// TIA Portal V20 export
FUNCTION_BLOCK "Sequence_1_SepaClamp"   // FB197, LAD
AUTHOR : ERsystem_FA2_DH. Kim
// stored: IsIECCheckEnabled true, MemoryReserve 100, Namespace Unit1.Em7, SetENOAutomatically false
   VAR
      statSelectedJobNumber { ExternalWritable := 'False'} : DInt;   // Evaluated Job Number
      instSequenceLADStatus { ExternalWritable := 'False'} : "LAF_StatusLadSequence";
      instSequenceLADControl { ExternalWritable := 'False'} : "LAF_ControlLadSequence";
      statTonTime { ExternalAccessible := 'False'; ExternalVisible := 'False'; ExternalWritable := 'False'} : Array[0..999] of TON_TIME;
   END_VAR
   VAR_TEMP
      tempCustomerAction : Bool;   // Placeholder for possible actions
      tempDo_nothing_and_wait_for_init : Bool;   // Placeholder for doing nothing
      tempSafeStateCondition : Bool;   // Temp Condition for the equipment module to be in a safe state
      tempIndex : Int;
   END_VAR
   VAR CONSTANT
      STEP_IDLE : DInt := 1;
      STEP_IMMEDIATE_STOP : DInt := 9001;   // Step executed when an immediate stop command is triggered for the sequence (i.e. when unit is in state aborting)
      JOB_1_STEP_01 : DInt := 101;
      JOB_1_STEP_10 : DInt := 110;
      JOB_1_STEP_20 : DInt := 120;
      JOB_1_STEP_30 : DInt := 130;
      JOB_1_STEP_80 : DInt := 180;
      JOB_1_STEP_90 : DInt := 190;
      JOB_2_STEP_01 : DInt := 201;
      JOB_2_STEP_10 : DInt := 210;
      JOB_2_STEP_11 : DInt := 211;
      JOB_2_STEP_20 : DInt := 220;
      JOB_2_STEP_21 : DInt := 221;
      JOB_2_STEP_30 : DInt := 230;
      JOB_2_STEP_40 : DInt := 240;
      JOB_2_STEP_41 : DInt := 241;
      JOB_2_STEP_50 : DInt := 250;
      JOB_2_STEP_51 : DInt := 251;
      JOB_2_STEP_60 : DInt := 260;
      JOB_2_STEP_80 : DInt := 280;
      JOB_2_STEP_90 : DInt := 290;
      JOB_3_STEP_01 : DInt := 301;
      JOB_3_STEP_10 : DInt := 310;
      JOB_3_STEP_11 : DInt := 311;
      JOB_3_STEP_20 : DInt := 320;
      JOB_3_STEP_21 : DInt := 321;
      JOB_3_STEP_22 : DInt := 322;
      JOB_3_STEP_23 : DInt := 323;
      JOB_3_STEP_24 : DInt := 324;
      JOB_3_STEP_30 : DInt := 330;
      JOB_3_STEP_31 : DInt := 331;
      JOB_3_STEP_40 : DInt := 340;
      JOB_3_STEP_80 : DInt := 380;
      JOB_3_STEP_90 : DInt := 390;
      JOB_4_STEP_01 : DInt := 401;
      JOB_4_STEP_10 : DInt := 410;
      JOB_4_STEP_11 : DInt := 411;
      JOB_4_STEP_90 : DInt := 490;
      JOB_5_STEP_01 : DInt := 501;
      JOB_5_STEP_10 : DInt := 510;
      JOB_5_STEP_11 : DInt := 511;
      JOB_5_STEP_20 : DInt := 520;
      JOB_5_STEP_21 : DInt := 521;
      JOB_5_STEP_30 : DInt := 530;
      JOB_5_STEP_90 : DInt := 590;
      JOB_6_STEP_01 : DInt := 601;
      JOB_6_STEP_10 : DInt := 610;
      JOB_6_STEP_11 : DInt := 611;
      JOB_6_STEP_20 : DInt := 620;
      JOB_6_STEP_30 : DInt := 630;
      JOB_6_STEP_90 : DInt := 690;
      JOB_10_STEP_01 : DInt := 1001;
      JOB_10_STEP_10 : DInt := 1010;
      JOB_10_STEP_11 : DInt := 1011;
      JOB_10_STEP_20 : DInt := 1020;
      JOB_10_STEP_90 : DInt := 1090;
      JOB_11_STEP_01 : DInt := 1101;
      JOB_11_STEP_10 : DInt := 1110;
      JOB_11_STEP_20 : DInt := 1120;
      JOB_11_STEP_30 : DInt := 1130;
      JOB_11_STEP_90 : DInt := 1190;
      JOB_12_STEP_01 : DInt := 1201;
      JOB_12_STEP_10 : DInt := 1210;
      JOB_12_STEP_20 : DInt := 1220;
      JOB_12_STEP_30 : DInt := 1230;
      JOB_12_STEP_40 : DInt := 1240;
      JOB_12_STEP_90 : DInt := 1290;
      FALSE : Bool := FALSE;
      TRUE : Bool := TRUE;
   END_VAR
   VAR_TEMP   // added for the SCL form of the ladder/FBD networks
      _w1 : Bool;
      _w2 : Bool;
   END_VAR
BEGIN

REGION Network 1: BLOCK INFO HEADER
   // (company) / (C) Copyright (year)
   // ---------------------------------------------------------------------------------
   // Title:                             (Title of this block)
   // Comment/Function: (that is implemented in the block)
   // Library/Family:           (that the source is dedicated to)
   // Author:                        (department / person in charge / contact)
   // Target System:          (test system with FW version)
   // Engineering:              TIA Portal (SW version)
   // Restrictions:               (OB types, etc.)
   // Requirements:           (hardware, technological package, etc.)
   // ---------------------------------------------------------------------------------
   // Change log table:
   // Version          | Date             | Signature      | Expert in charge  | Changes applied ------------------------|----------------------|-------------------------|--------------------------------|-----------------------
   // 001.000.000 | yyyy-mm-dd | 0x00000000 | (name of expert) | First released version
END_REGION

REGION Network 2: DESCRIPTION
   // This is a template block provided by the Automation Framework. It can be used to create an own project.
   // The Block Info Header is prepared to put in your own data.
   // Description of the block could be added here and the docu created by Code2Docu.
END_REGION

REGION Network 3: ********************* CONTROL *************************
END_REGION

REGION Network 4: Sequence Control
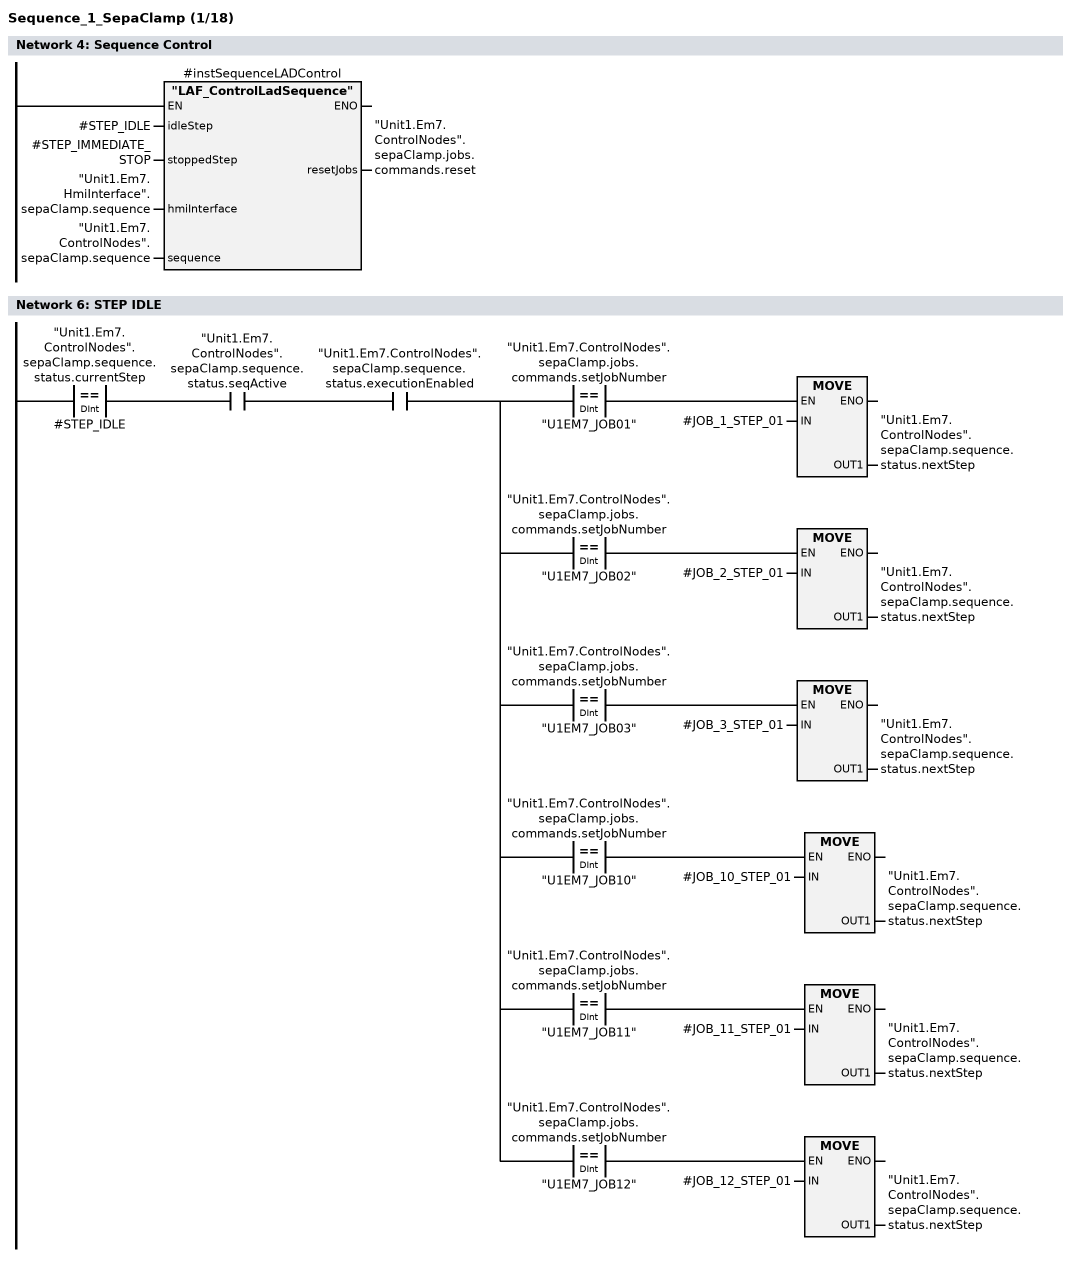
   RUNG wire#powerrail
      #instSequenceLADControl(idleStep := #STEP_IDLE, stoppedStep := #STEP_IMMEDIATE_STOP, hmiInterface := "Unit1.Em7.HmiInterface".sepaClamp.sequence, sequence := "Unit1.Em7.ControlNodes".sepaClamp.sequence, resetJobs => "Unit1.Em7.ControlNodes".sepaClamp.jobs.commands.reset)
   END_RUNG
   // the same network as SCL:
   #instSequenceLADControl(idleStep := #STEP_IDLE,   // "LAF_ControlLadSequence"
                           stoppedStep := #STEP_IMMEDIATE_STOP,
                           hmiInterface := "Unit1.Em7.HmiInterface".sepaClamp.sequence,
                           sequence := "Unit1.Em7.ControlNodes".sepaClamp.sequence,
                           resetJobs => "Unit1.Em7.ControlNodes".sepaClamp.jobs.commands.reset);
END_REGION

REGION Network 5: *************** JOB SELECT **************************
END_REGION

REGION Network 6: STEP IDLE
   RUNG wire#powerrail
      { S7_Templates := "SrcType := DInt" } EQ_Contact(in1 := "Unit1.Em7.ControlNodes".sepaClamp.sequence.status.currentStep, in2 := #STEP_IDLE)
      Contact( "Unit1.Em7.ControlNodes".sepaClamp.sequence.status.seqActive )
      Contact( "Unit1.Em7.ControlNodes".sepaClamp.sequence.status.executionEnabled )
      wire#w1
      { S7_Templates := "SrcType := DInt" } EQ_Contact(in1 := "Unit1.Em7.ControlNodes".sepaClamp.jobs.commands.setJobNumber, in2 := "U1EM7_JOB01")
      Move(in := #JOB_1_STEP_01, out1 => "Unit1.Em7.ControlNodes".sepaClamp.sequence.status.nextStep)
   END_RUNG
   RUNG wire#w1
      { S7_Templates := "SrcType := DInt" } EQ_Contact(in1 := "Unit1.Em7.ControlNodes".sepaClamp.jobs.commands.setJobNumber, in2 := "U1EM7_JOB02")
      Move(in := #JOB_2_STEP_01, out1 => "Unit1.Em7.ControlNodes".sepaClamp.sequence.status.nextStep)
   END_RUNG
   RUNG wire#w1
      { S7_Templates := "SrcType := DInt" } EQ_Contact(in1 := "Unit1.Em7.ControlNodes".sepaClamp.jobs.commands.setJobNumber, in2 := "U1EM7_JOB03")
      Move(in := #JOB_3_STEP_01, out1 => "Unit1.Em7.ControlNodes".sepaClamp.sequence.status.nextStep)
   END_RUNG
   RUNG wire#w1
      { S7_Templates := "SrcType := DInt" } EQ_Contact(in1 := "Unit1.Em7.ControlNodes".sepaClamp.jobs.commands.setJobNumber, in2 := "U1EM7_JOB10")
      Move(in := #JOB_10_STEP_01, out1 => "Unit1.Em7.ControlNodes".sepaClamp.sequence.status.nextStep)
   END_RUNG
   RUNG wire#w1
      { S7_Templates := "SrcType := DInt" } EQ_Contact(in1 := "Unit1.Em7.ControlNodes".sepaClamp.jobs.commands.setJobNumber, in2 := "U1EM7_JOB11")
      Move(in := #JOB_11_STEP_01, out1 => "Unit1.Em7.ControlNodes".sepaClamp.sequence.status.nextStep)
   END_RUNG
   RUNG wire#w1
      { S7_Templates := "SrcType := DInt" } EQ_Contact(in1 := "Unit1.Em7.ControlNodes".sepaClamp.jobs.commands.setJobNumber, in2 := "U1EM7_JOB12")
      Move(in := #JOB_12_STEP_01, out1 => "Unit1.Em7.ControlNodes".sepaClamp.sequence.status.nextStep)
   END_RUNG
   // the same network as SCL:
   #_w1 := ("Unit1.Em7.ControlNodes".sepaClamp.sequence.status.currentStep = #STEP_IDLE) AND "Unit1.Em7.ControlNodes".sepaClamp.sequence.status.seqActive AND "Unit1.Em7.ControlNodes".sepaClamp.sequence.status.executionEnabled;
   IF #_w1 AND ("Unit1.Em7.ControlNodes".sepaClamp.jobs.commands.setJobNumber = "U1EM7_JOB01") THEN
       "Unit1.Em7.ControlNodes".sepaClamp.sequence.status.nextStep := #JOB_1_STEP_01;
   END_IF;
   IF #_w1 AND ("Unit1.Em7.ControlNodes".sepaClamp.jobs.commands.setJobNumber = "U1EM7_JOB02") THEN
       "Unit1.Em7.ControlNodes".sepaClamp.sequence.status.nextStep := #JOB_2_STEP_01;
   END_IF;
   IF #_w1 AND ("Unit1.Em7.ControlNodes".sepaClamp.jobs.commands.setJobNumber = "U1EM7_JOB03") THEN
       "Unit1.Em7.ControlNodes".sepaClamp.sequence.status.nextStep := #JOB_3_STEP_01;
   END_IF;
   IF #_w1 AND ("Unit1.Em7.ControlNodes".sepaClamp.jobs.commands.setJobNumber = "U1EM7_JOB10") THEN
       "Unit1.Em7.ControlNodes".sepaClamp.sequence.status.nextStep := #JOB_10_STEP_01;
   END_IF;
   IF #_w1 AND ("Unit1.Em7.ControlNodes".sepaClamp.jobs.commands.setJobNumber = "U1EM7_JOB11") THEN
       "Unit1.Em7.ControlNodes".sepaClamp.sequence.status.nextStep := #JOB_11_STEP_01;
   END_IF;
   IF #_w1 AND ("Unit1.Em7.ControlNodes".sepaClamp.jobs.commands.setJobNumber = "U1EM7_JOB12") THEN
       "Unit1.Em7.ControlNodes".sepaClamp.sequence.status.nextStep := #JOB_12_STEP_01;
   END_IF;
END_REGION

REGION Network 7: *************** JOB[1] EM HOMING ************************
END_REGION

REGION Network 8: Step[101] : JOB[1] Condition
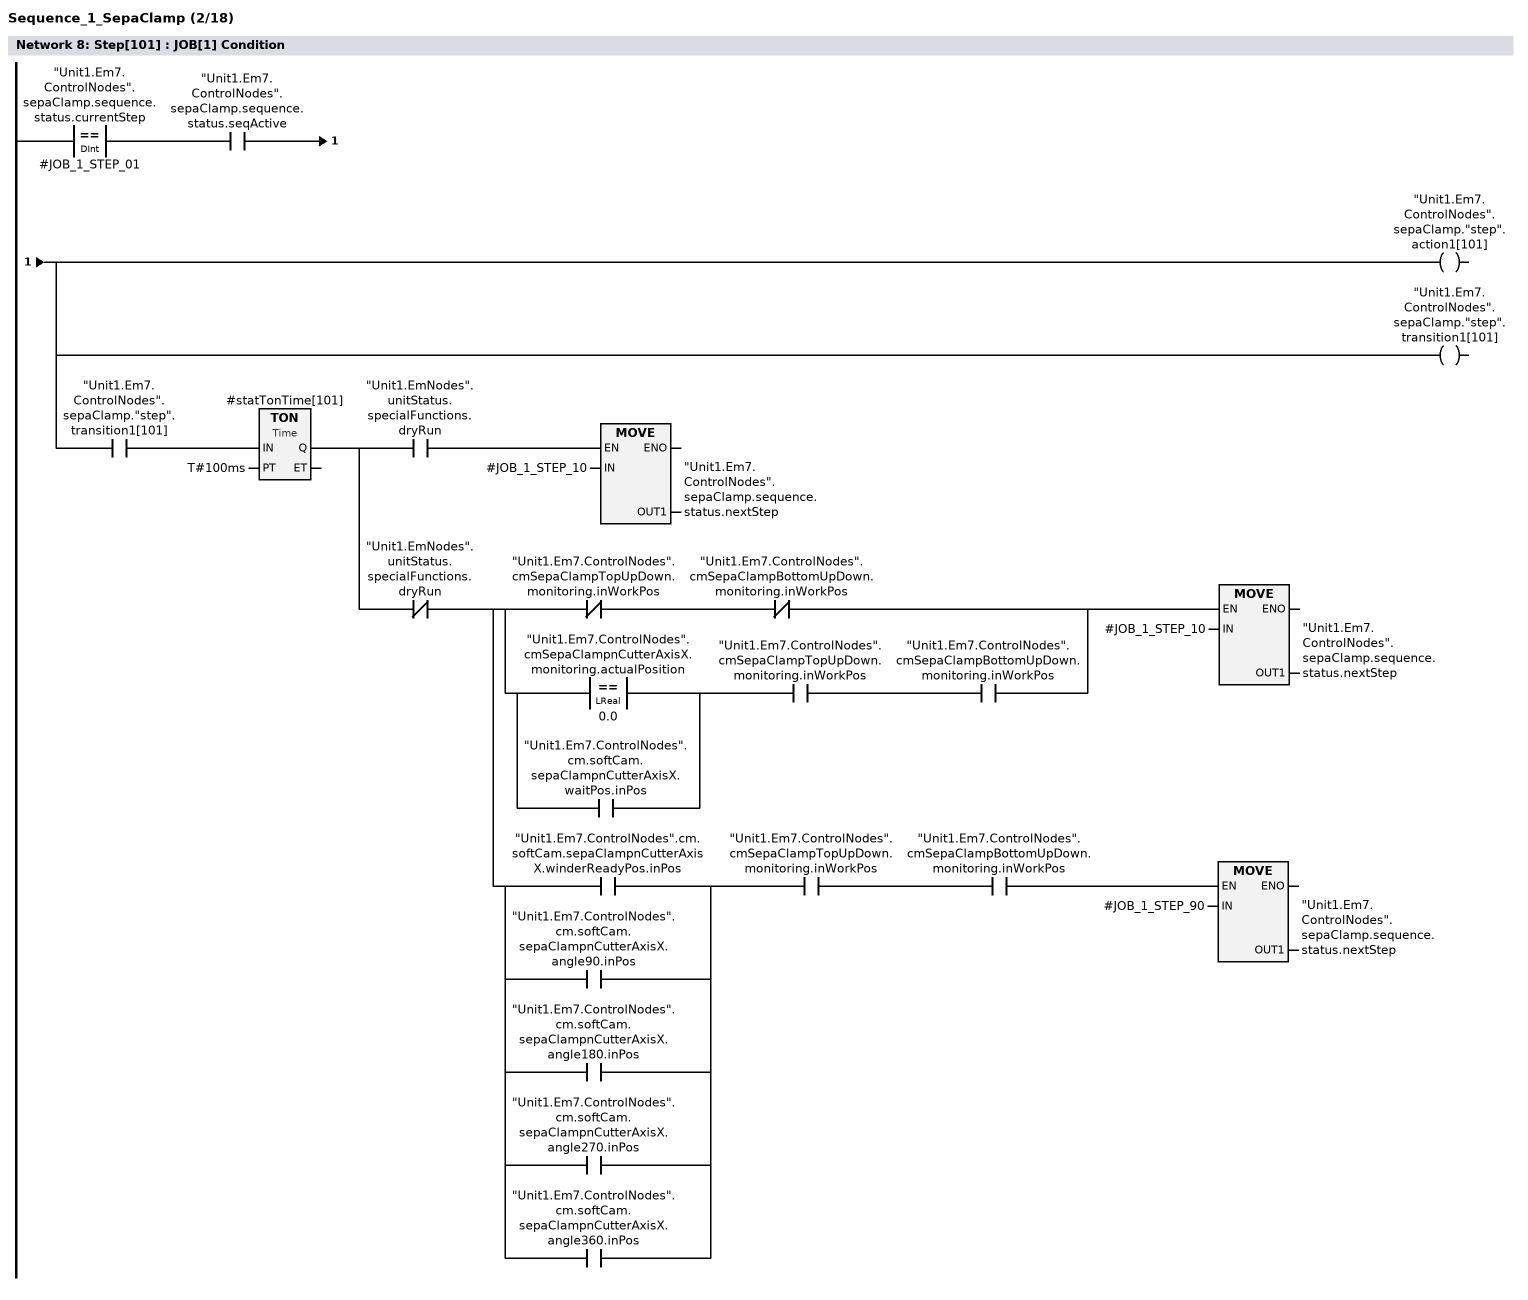
   RUNG wire#powerrail
      { S7_Templates := "SrcType := DInt" } EQ_Contact(in1 := "Unit1.Em7.ControlNodes".sepaClamp.sequence.status.currentStep, in2 := #JOB_1_STEP_01)
      Contact( "Unit1.Em7.ControlNodes".sepaClamp.sequence.status.seqActive )
      wire#w1
      Coil( "Unit1.Em7.ControlNodes".sepaClamp."step".action1[101] )
   END_RUNG
   RUNG wire#w1
      Coil( "Unit1.Em7.ControlNodes".sepaClamp."step".transition1[101] )
   END_RUNG
   RUNG wire#w1
      Contact( "Unit1.Em7.ControlNodes".sepaClamp."step".transition1[101] )
      { S7_Templates := "time_type := Time" } #statTonTime[101].TON(pt := T#100ms, et =>)
      wire#w2
      Contact( "Unit1.EmNodes".unitStatus.specialFunctions.dryRun )
      Move(in := #JOB_1_STEP_10, out1 => "Unit1.Em7.ControlNodes".sepaClamp.sequence.status.nextStep)
   END_RUNG
   RUNG wire#w2
      I_Contact( "Unit1.EmNodes".unitStatus.specialFunctions.dryRun )
      wire#w3
      I_Contact( "Unit1.Em7.ControlNodes".cmSepaClampTopUpDown.monitoring.inWorkPos )
      I_Contact( "Unit1.Em7.ControlNodes".cmSepaClampBottomUpDown.monitoring.inWorkPos )
      wire#w4
      Move(in := #JOB_1_STEP_10, out1 => "Unit1.Em7.ControlNodes".sepaClamp.sequence.status.nextStep)
   END_RUNG
   RUNG wire#w3
      { S7_Templates := "SrcType := LReal" } EQ_Contact(in1 := "Unit1.Em7.ControlNodes".cmSepaClampnCutterAxisX.monitoring.actualPosition, in2 := 0.0)
      wire#w5
      Contact( "Unit1.Em7.ControlNodes".cmSepaClampTopUpDown.monitoring.inWorkPos )
      Contact( "Unit1.Em7.ControlNodes".cmSepaClampBottomUpDown.monitoring.inWorkPos )
   END_RUNG wire#w4
   RUNG wire#w3
      Contact( "Unit1.Em7.ControlNodes".cm.softCam.sepaClampnCutterAxisX.waitPos.inPos )
   END_RUNG wire#w5
   RUNG wire#w3
      Contact( "Unit1.Em7.ControlNodes".cm.softCam.sepaClampnCutterAxisX.winderReadyPos.inPos )
      wire#w6
      Contact( "Unit1.Em7.ControlNodes".cmSepaClampTopUpDown.monitoring.inWorkPos )
      Contact( "Unit1.Em7.ControlNodes".cmSepaClampBottomUpDown.monitoring.inWorkPos )
      Move(in := #JOB_1_STEP_90, out1 => "Unit1.Em7.ControlNodes".sepaClamp.sequence.status.nextStep)
   END_RUNG
   RUNG wire#w3
      Contact( "Unit1.Em7.ControlNodes".cm.softCam.sepaClampnCutterAxisX.angle90.inPos )
   END_RUNG wire#w6
   RUNG wire#w3
      Contact( "Unit1.Em7.ControlNodes".cm.softCam.sepaClampnCutterAxisX.angle180.inPos )
   END_RUNG wire#w6
   RUNG wire#w3
      Contact( "Unit1.Em7.ControlNodes".cm.softCam.sepaClampnCutterAxisX.angle270.inPos )
   END_RUNG wire#w6
   RUNG wire#w3
      Contact( "Unit1.Em7.ControlNodes".cm.softCam.sepaClampnCutterAxisX.angle360.inPos )
   END_RUNG wire#w6
   // the same network as SCL:
   "Unit1.Em7.ControlNodes".sepaClamp."step".action1[101] := ("Unit1.Em7.ControlNodes".sepaClamp.sequence.status.currentStep = #JOB_1_STEP_01) AND "Unit1.Em7.ControlNodes".sepaClamp.sequence.status.seqActive;
   "Unit1.Em7.ControlNodes".sepaClamp."step".transition1[101] := ("Unit1.Em7.ControlNodes".sepaClamp.sequence.status.currentStep = #JOB_1_STEP_01) AND "Unit1.Em7.ControlNodes".sepaClamp.sequence.status.seqActive;
   #statTonTime[101].TON(IN := ("Unit1.Em7.ControlNodes".sepaClamp.sequence.status.currentStep = #JOB_1_STEP_01) AND "Unit1.Em7.ControlNodes".sepaClamp.sequence.status.seqActive AND "Unit1.Em7.ControlNodes".sepaClamp."step".transition1[101],
                         PT := T#100ms);
   IF #statTonTime[101].Q AND "Unit1.EmNodes".unitStatus.specialFunctions.dryRun THEN
       "Unit1.Em7.ControlNodes".sepaClamp.sequence.status.nextStep := #JOB_1_STEP_10;
   END_IF;
   #_w1 := #statTonTime[101].Q AND NOT "Unit1.EmNodes".unitStatus.specialFunctions.dryRun;
   IF #_w1 AND ((NOT "Unit1.Em7.ControlNodes".cmSepaClampTopUpDown.monitoring.inWorkPos AND NOT "Unit1.Em7.ControlNodes".cmSepaClampBottomUpDown.monitoring.inWorkPos) OR ((("Unit1.Em7.ControlNodes".cmSepaClampnCutterAxisX.monitoring.actualPosition = 0.0) OR "Unit1.Em7.ControlNodes".cm.softCam.sepaClampnCutterAxisX.waitPos.inPos) AND "Unit1.Em7.ControlNodes".cmSepaClampTopUpDown.monitoring.inWorkPos AND "Unit1.Em7.ControlNodes".cmSepaClampBottomUpDown.monitoring.inWorkPos)) THEN
       "Unit1.Em7.ControlNodes".sepaClamp.sequence.status.nextStep := #JOB_1_STEP_10;
   END_IF;
   IF #_w1 AND ("Unit1.Em7.ControlNodes".cm.softCam.sepaClampnCutterAxisX.winderReadyPos.inPos OR "Unit1.Em7.ControlNodes".cm.softCam.sepaClampnCutterAxisX.angle90.inPos OR "Unit1.Em7.ControlNodes".cm.softCam.sepaClampnCutterAxisX.angle180.inPos OR "Unit1.Em7.ControlNodes".cm.softCam.sepaClampnCutterAxisX.angle270.inPos OR "Unit1.Em7.ControlNodes".cm.softCam.sepaClampnCutterAxisX.angle360.inPos) AND "Unit1.Em7.ControlNodes".cmSepaClampTopUpDown.monitoring.inWorkPos AND "Unit1.Em7.ControlNodes".cmSepaClampBottomUpDown.monitoring.inWorkPos THEN
       "Unit1.Em7.ControlNodes".sepaClamp.sequence.status.nextStep := #JOB_1_STEP_90;
   END_IF;
END_REGION

REGION Network 9: Step[110] : Cutter Up
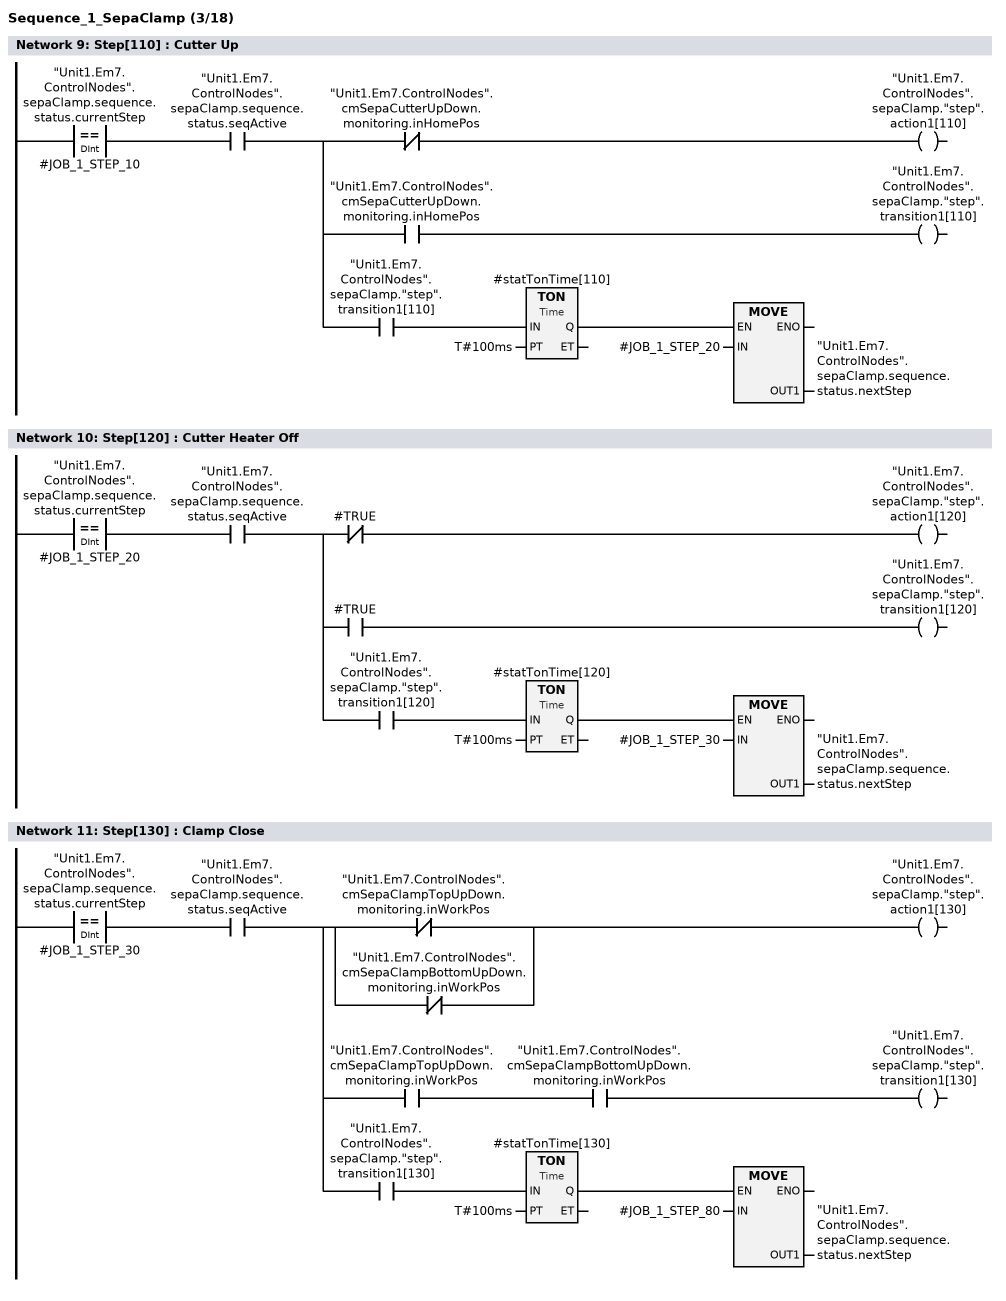
   RUNG wire#powerrail
      { S7_Templates := "SrcType := DInt" } EQ_Contact(in1 := "Unit1.Em7.ControlNodes".sepaClamp.sequence.status.currentStep, in2 := #JOB_1_STEP_10)
      Contact( "Unit1.Em7.ControlNodes".sepaClamp.sequence.status.seqActive )
      wire#w1
      I_Contact( "Unit1.Em7.ControlNodes".cmSepaCutterUpDown.monitoring.inHomePos )
      Coil( "Unit1.Em7.ControlNodes".sepaClamp."step".action1[110] )
   END_RUNG
   RUNG wire#w1
      Contact( "Unit1.Em7.ControlNodes".cmSepaCutterUpDown.monitoring.inHomePos )
      Coil( "Unit1.Em7.ControlNodes".sepaClamp."step".transition1[110] )
   END_RUNG
   RUNG wire#w1
      Contact( "Unit1.Em7.ControlNodes".sepaClamp."step".transition1[110] )
      { S7_Templates := "time_type := Time" } #statTonTime[110].TON(pt := T#100ms, et =>)
      Move(in := #JOB_1_STEP_20, out1 => "Unit1.Em7.ControlNodes".sepaClamp.sequence.status.nextStep)
   END_RUNG
   // the same network as SCL:
   #_w1 := ("Unit1.Em7.ControlNodes".sepaClamp.sequence.status.currentStep = #JOB_1_STEP_10) AND "Unit1.Em7.ControlNodes".sepaClamp.sequence.status.seqActive;
   "Unit1.Em7.ControlNodes".sepaClamp."step".action1[110] := #_w1 AND NOT "Unit1.Em7.ControlNodes".cmSepaCutterUpDown.monitoring.inHomePos;
   "Unit1.Em7.ControlNodes".sepaClamp."step".transition1[110] := #_w1 AND "Unit1.Em7.ControlNodes".cmSepaCutterUpDown.monitoring.inHomePos;
   #statTonTime[110].TON(IN := #_w1 AND "Unit1.Em7.ControlNodes".sepaClamp."step".transition1[110],
                         PT := T#100ms);
   IF #statTonTime[110].Q THEN
       "Unit1.Em7.ControlNodes".sepaClamp.sequence.status.nextStep := #JOB_1_STEP_20;
   END_IF;
END_REGION

REGION Network 10: Step[120] : Cutter Heater Off
   RUNG wire#powerrail
      { S7_Templates := "SrcType := DInt" } EQ_Contact(in1 := "Unit1.Em7.ControlNodes".sepaClamp.sequence.status.currentStep, in2 := #JOB_1_STEP_20)
      Contact( "Unit1.Em7.ControlNodes".sepaClamp.sequence.status.seqActive )
      wire#w1
      I_Contact( #TRUE )
      Coil( "Unit1.Em7.ControlNodes".sepaClamp."step".action1[120] )
   END_RUNG
   RUNG wire#w1
      Contact( #TRUE )
      Coil( "Unit1.Em7.ControlNodes".sepaClamp."step".transition1[120] )
   END_RUNG
   RUNG wire#w1
      Contact( "Unit1.Em7.ControlNodes".sepaClamp."step".transition1[120] )
      { S7_Templates := "time_type := Time" } #statTonTime[120].TON(pt := T#100ms, et =>)
      Move(in := #JOB_1_STEP_30, out1 => "Unit1.Em7.ControlNodes".sepaClamp.sequence.status.nextStep)
   END_RUNG
   // the same network as SCL:
   #_w1 := ("Unit1.Em7.ControlNodes".sepaClamp.sequence.status.currentStep = #JOB_1_STEP_20) AND "Unit1.Em7.ControlNodes".sepaClamp.sequence.status.seqActive;
   "Unit1.Em7.ControlNodes".sepaClamp."step".action1[120] := #_w1 AND NOT #TRUE;
   "Unit1.Em7.ControlNodes".sepaClamp."step".transition1[120] := #_w1 AND #TRUE;
   #statTonTime[120].TON(IN := #_w1 AND "Unit1.Em7.ControlNodes".sepaClamp."step".transition1[120],
                         PT := T#100ms);
   IF #statTonTime[120].Q THEN
       "Unit1.Em7.ControlNodes".sepaClamp.sequence.status.nextStep := #JOB_1_STEP_30;
   END_IF;
END_REGION

REGION Network 11: Step[130] : Clamp Close
   RUNG wire#powerrail
      { S7_Templates := "SrcType := DInt" } EQ_Contact(in1 := "Unit1.Em7.ControlNodes".sepaClamp.sequence.status.currentStep, in2 := #JOB_1_STEP_30)
      Contact( "Unit1.Em7.ControlNodes".sepaClamp.sequence.status.seqActive )
      wire#w1
      I_Contact( "Unit1.Em7.ControlNodes".cmSepaClampTopUpDown.monitoring.inWorkPos )
      wire#w2
      Coil( "Unit1.Em7.ControlNodes".sepaClamp."step".action1[130] )
   END_RUNG
   RUNG wire#w1
      I_Contact( "Unit1.Em7.ControlNodes".cmSepaClampBottomUpDown.monitoring.inWorkPos )
   END_RUNG wire#w2
   RUNG wire#w1
      Contact( "Unit1.Em7.ControlNodes".cmSepaClampTopUpDown.monitoring.inWorkPos )
      Contact( "Unit1.Em7.ControlNodes".cmSepaClampBottomUpDown.monitoring.inWorkPos )
      Coil( "Unit1.Em7.ControlNodes".sepaClamp."step".transition1[130] )
   END_RUNG
   RUNG wire#w1
      Contact( "Unit1.Em7.ControlNodes".sepaClamp."step".transition1[130] )
      { S7_Templates := "time_type := Time" } #statTonTime[130].TON(pt := T#100ms, et =>)
      Move(in := #JOB_1_STEP_80, out1 => "Unit1.Em7.ControlNodes".sepaClamp.sequence.status.nextStep)
   END_RUNG
   // the same network as SCL:
   #_w1 := ("Unit1.Em7.ControlNodes".sepaClamp.sequence.status.currentStep = #JOB_1_STEP_30) AND "Unit1.Em7.ControlNodes".sepaClamp.sequence.status.seqActive;
   "Unit1.Em7.ControlNodes".sepaClamp."step".action1[130] := #_w1 AND (NOT "Unit1.Em7.ControlNodes".cmSepaClampTopUpDown.monitoring.inWorkPos OR NOT "Unit1.Em7.ControlNodes".cmSepaClampBottomUpDown.monitoring.inWorkPos);
   "Unit1.Em7.ControlNodes".sepaClamp."step".transition1[130] := #_w1 AND "Unit1.Em7.ControlNodes".cmSepaClampTopUpDown.monitoring.inWorkPos AND "Unit1.Em7.ControlNodes".cmSepaClampBottomUpDown.monitoring.inWorkPos;
   #statTonTime[130].TON(IN := #_w1 AND "Unit1.Em7.ControlNodes".sepaClamp."step".transition1[130],
                         PT := T#100ms);
   IF #statTonTime[130].Q THEN
       "Unit1.Em7.ControlNodes".sepaClamp.sequence.status.nextStep := #JOB_1_STEP_80;
   END_IF;
END_REGION

REGION Network 12: Step[180] : Clamp X,Z-Axis Wait Pos
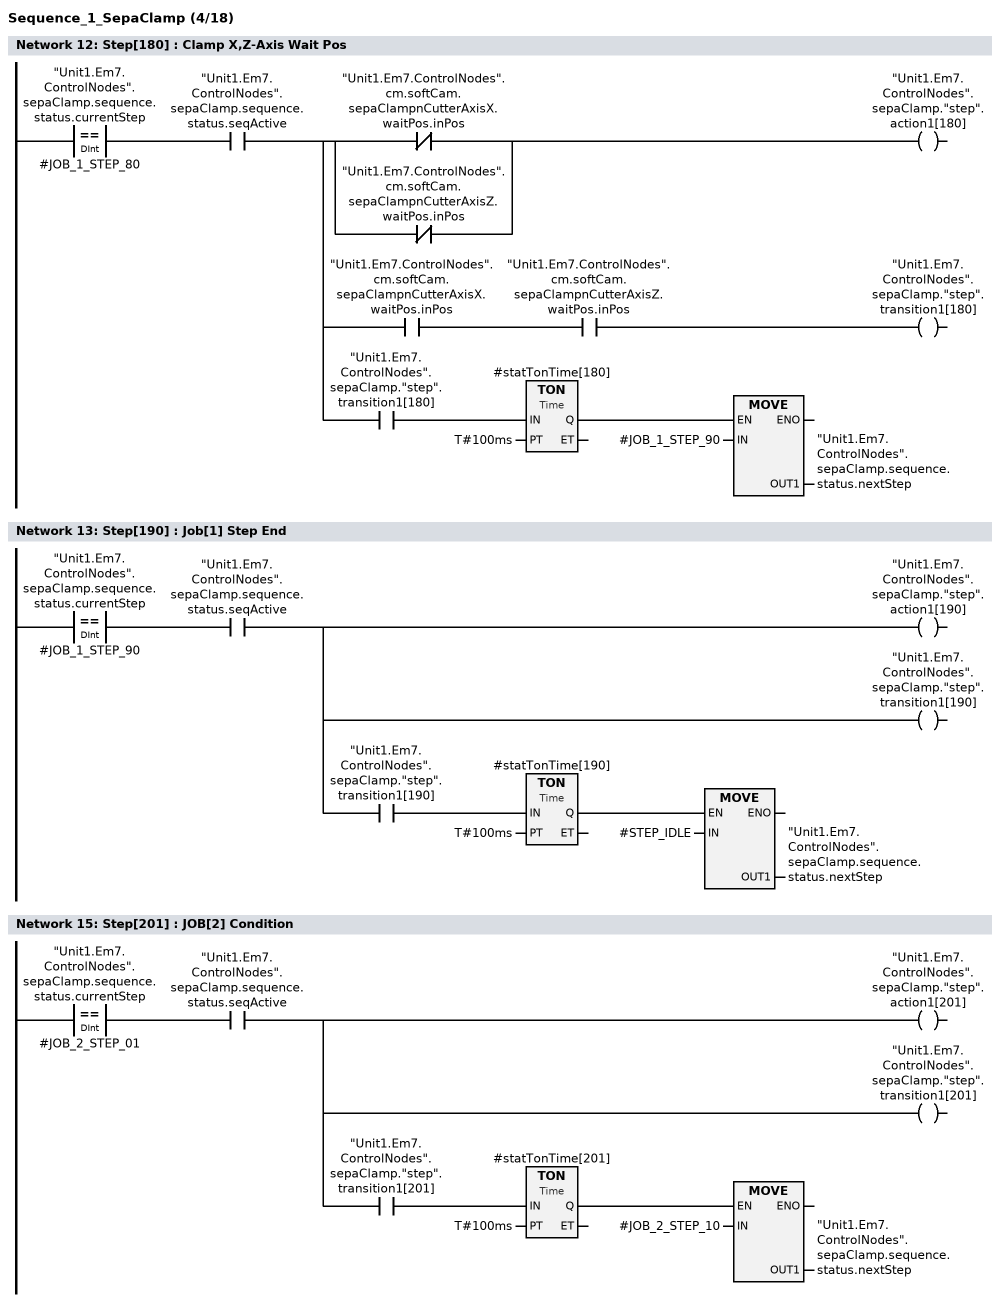
   RUNG wire#powerrail
      { S7_Templates := "SrcType := DInt" } EQ_Contact(in1 := "Unit1.Em7.ControlNodes".sepaClamp.sequence.status.currentStep, in2 := #JOB_1_STEP_80)
      Contact( "Unit1.Em7.ControlNodes".sepaClamp.sequence.status.seqActive )
      wire#w1
      I_Contact( "Unit1.Em7.ControlNodes".cm.softCam.sepaClampnCutterAxisX.waitPos.inPos )
      wire#w2
      Coil( "Unit1.Em7.ControlNodes".sepaClamp."step".action1[180] )
   END_RUNG
   RUNG wire#w1
      I_Contact( "Unit1.Em7.ControlNodes".cm.softCam.sepaClampnCutterAxisZ.waitPos.inPos )
   END_RUNG wire#w2
   RUNG wire#w1
      Contact( "Unit1.Em7.ControlNodes".cm.softCam.sepaClampnCutterAxisX.waitPos.inPos )
      Contact( "Unit1.Em7.ControlNodes".cm.softCam.sepaClampnCutterAxisZ.waitPos.inPos )
      Coil( "Unit1.Em7.ControlNodes".sepaClamp."step".transition1[180] )
   END_RUNG
   RUNG wire#w1
      Contact( "Unit1.Em7.ControlNodes".sepaClamp."step".transition1[180] )
      { S7_Templates := "time_type := Time" } #statTonTime[180].TON(pt := T#100ms, et =>)
      Move(in := #JOB_1_STEP_90, out1 => "Unit1.Em7.ControlNodes".sepaClamp.sequence.status.nextStep)
   END_RUNG
   // the same network as SCL:
   #_w1 := ("Unit1.Em7.ControlNodes".sepaClamp.sequence.status.currentStep = #JOB_1_STEP_80) AND "Unit1.Em7.ControlNodes".sepaClamp.sequence.status.seqActive;
   "Unit1.Em7.ControlNodes".sepaClamp."step".action1[180] := #_w1 AND (NOT "Unit1.Em7.ControlNodes".cm.softCam.sepaClampnCutterAxisX.waitPos.inPos OR NOT "Unit1.Em7.ControlNodes".cm.softCam.sepaClampnCutterAxisZ.waitPos.inPos);
   "Unit1.Em7.ControlNodes".sepaClamp."step".transition1[180] := #_w1 AND "Unit1.Em7.ControlNodes".cm.softCam.sepaClampnCutterAxisX.waitPos.inPos AND "Unit1.Em7.ControlNodes".cm.softCam.sepaClampnCutterAxisZ.waitPos.inPos;
   #statTonTime[180].TON(IN := #_w1 AND "Unit1.Em7.ControlNodes".sepaClamp."step".transition1[180],
                         PT := T#100ms);
   IF #statTonTime[180].Q THEN
       "Unit1.Em7.ControlNodes".sepaClamp.sequence.status.nextStep := #JOB_1_STEP_90;
   END_IF;
END_REGION

REGION Network 13: Step[190] : Job[1] Step End
   RUNG wire#powerrail
      { S7_Templates := "SrcType := DInt" } EQ_Contact(in1 := "Unit1.Em7.ControlNodes".sepaClamp.sequence.status.currentStep, in2 := #JOB_1_STEP_90)
      Contact( "Unit1.Em7.ControlNodes".sepaClamp.sequence.status.seqActive )
      wire#w1
      Coil( "Unit1.Em7.ControlNodes".sepaClamp."step".action1[190] )
   END_RUNG
   RUNG wire#w1
      Coil( "Unit1.Em7.ControlNodes".sepaClamp."step".transition1[190] )
   END_RUNG
   RUNG wire#w1
      Contact( "Unit1.Em7.ControlNodes".sepaClamp."step".transition1[190] )
      { S7_Templates := "time_type := Time" } #statTonTime[190].TON(pt := T#100ms, et =>)
      Move(in := #STEP_IDLE, out1 => "Unit1.Em7.ControlNodes".sepaClamp.sequence.status.nextStep)
   END_RUNG
   // the same network as SCL:
   "Unit1.Em7.ControlNodes".sepaClamp."step".action1[190] := ("Unit1.Em7.ControlNodes".sepaClamp.sequence.status.currentStep = #JOB_1_STEP_90) AND "Unit1.Em7.ControlNodes".sepaClamp.sequence.status.seqActive;
   "Unit1.Em7.ControlNodes".sepaClamp."step".transition1[190] := ("Unit1.Em7.ControlNodes".sepaClamp.sequence.status.currentStep = #JOB_1_STEP_90) AND "Unit1.Em7.ControlNodes".sepaClamp.sequence.status.seqActive;
   #statTonTime[190].TON(IN := ("Unit1.Em7.ControlNodes".sepaClamp.sequence.status.currentStep = #JOB_1_STEP_90) AND "Unit1.Em7.ControlNodes".sepaClamp.sequence.status.seqActive AND "Unit1.Em7.ControlNodes".sepaClamp."step".transition1[190],
                         PT := T#100ms);
   IF #statTonTime[190].Q THEN
       "Unit1.Em7.ControlNodes".sepaClamp.sequence.status.nextStep := #STEP_IDLE;
   END_IF;
END_REGION

REGION Network 14: ******************** JOB[2] Load ********************
END_REGION

REGION Network 15: Step[201] : JOB[2] Condition
   RUNG wire#powerrail
      { S7_Templates := "SrcType := DInt" } EQ_Contact(in1 := "Unit1.Em7.ControlNodes".sepaClamp.sequence.status.currentStep, in2 := #JOB_2_STEP_01)
      Contact( "Unit1.Em7.ControlNodes".sepaClamp.sequence.status.seqActive )
      wire#w1
      Coil( "Unit1.Em7.ControlNodes".sepaClamp."step".action1[201] )
   END_RUNG
   RUNG wire#w1
      Coil( "Unit1.Em7.ControlNodes".sepaClamp."step".transition1[201] )
   END_RUNG
   RUNG wire#w1
      Contact( "Unit1.Em7.ControlNodes".sepaClamp."step".transition1[201] )
      { S7_Templates := "time_type := Time" } #statTonTime[201].TON(pt := T#100ms, et =>)
      Move(in := #JOB_2_STEP_10, out1 => "Unit1.Em7.ControlNodes".sepaClamp.sequence.status.nextStep)
   END_RUNG
   // the same network as SCL:
   "Unit1.Em7.ControlNodes".sepaClamp."step".action1[201] := ("Unit1.Em7.ControlNodes".sepaClamp.sequence.status.currentStep = #JOB_2_STEP_01) AND "Unit1.Em7.ControlNodes".sepaClamp.sequence.status.seqActive;
   "Unit1.Em7.ControlNodes".sepaClamp."step".transition1[201] := ("Unit1.Em7.ControlNodes".sepaClamp.sequence.status.currentStep = #JOB_2_STEP_01) AND "Unit1.Em7.ControlNodes".sepaClamp.sequence.status.seqActive;
   #statTonTime[201].TON(IN := ("Unit1.Em7.ControlNodes".sepaClamp.sequence.status.currentStep = #JOB_2_STEP_01) AND "Unit1.Em7.ControlNodes".sepaClamp.sequence.status.seqActive AND "Unit1.Em7.ControlNodes".sepaClamp."step".transition1[201],
                         PT := T#100ms);
   IF #statTonTime[201].Q THEN
       "Unit1.Em7.ControlNodes".sepaClamp.sequence.status.nextStep := #JOB_2_STEP_10;
   END_IF;
END_REGION

REGION Network 16: Step[210] : Clamp X,Z-Axis Load Pos
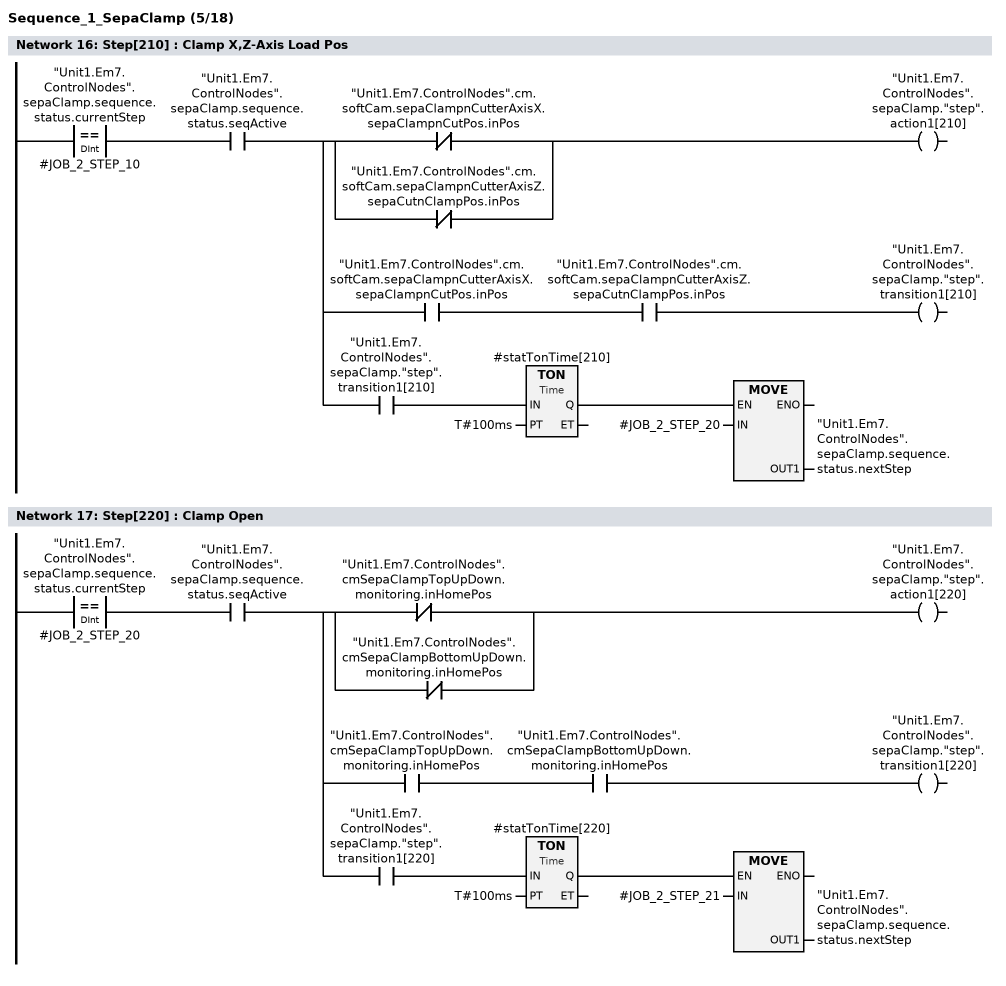
   RUNG wire#powerrail
      { S7_Templates := "SrcType := DInt" } EQ_Contact(in1 := "Unit1.Em7.ControlNodes".sepaClamp.sequence.status.currentStep, in2 := #JOB_2_STEP_10)
      Contact( "Unit1.Em7.ControlNodes".sepaClamp.sequence.status.seqActive )
      wire#w1
      I_Contact( "Unit1.Em7.ControlNodes".cm.softCam.sepaClampnCutterAxisX.sepaClampnCutPos.inPos )
      wire#w2
      Coil( "Unit1.Em7.ControlNodes".sepaClamp."step".action1[210] )
   END_RUNG
   RUNG wire#w1
      I_Contact( "Unit1.Em7.ControlNodes".cm.softCam.sepaClampnCutterAxisZ.sepaCutnClampPos.inPos )
   END_RUNG wire#w2
   RUNG wire#w1
      Contact( "Unit1.Em7.ControlNodes".cm.softCam.sepaClampnCutterAxisX.sepaClampnCutPos.inPos )
      Contact( "Unit1.Em7.ControlNodes".cm.softCam.sepaClampnCutterAxisZ.sepaCutnClampPos.inPos )
      Coil( "Unit1.Em7.ControlNodes".sepaClamp."step".transition1[210] )
   END_RUNG
   RUNG wire#w1
      Contact( "Unit1.Em7.ControlNodes".sepaClamp."step".transition1[210] )
      { S7_Templates := "time_type := Time" } #statTonTime[210].TON(pt := T#100ms, et =>)
      Move(in := #JOB_2_STEP_20, out1 => "Unit1.Em7.ControlNodes".sepaClamp.sequence.status.nextStep)
   END_RUNG
   // the same network as SCL:
   #_w1 := ("Unit1.Em7.ControlNodes".sepaClamp.sequence.status.currentStep = #JOB_2_STEP_10) AND "Unit1.Em7.ControlNodes".sepaClamp.sequence.status.seqActive;
   "Unit1.Em7.ControlNodes".sepaClamp."step".action1[210] := #_w1 AND (NOT "Unit1.Em7.ControlNodes".cm.softCam.sepaClampnCutterAxisX.sepaClampnCutPos.inPos OR NOT "Unit1.Em7.ControlNodes".cm.softCam.sepaClampnCutterAxisZ.sepaCutnClampPos.inPos);
   "Unit1.Em7.ControlNodes".sepaClamp."step".transition1[210] := #_w1 AND "Unit1.Em7.ControlNodes".cm.softCam.sepaClampnCutterAxisX.sepaClampnCutPos.inPos AND "Unit1.Em7.ControlNodes".cm.softCam.sepaClampnCutterAxisZ.sepaCutnClampPos.inPos;
   #statTonTime[210].TON(IN := #_w1 AND "Unit1.Em7.ControlNodes".sepaClamp."step".transition1[210],
                         PT := T#100ms);
   IF #statTonTime[210].Q THEN
       "Unit1.Em7.ControlNodes".sepaClamp.sequence.status.nextStep := #JOB_2_STEP_20;
   END_IF;
END_REGION

REGION Network 17: Step[220] : Clamp Open
   RUNG wire#powerrail
      { S7_Templates := "SrcType := DInt" } EQ_Contact(in1 := "Unit1.Em7.ControlNodes".sepaClamp.sequence.status.currentStep, in2 := #JOB_2_STEP_20)
      Contact( "Unit1.Em7.ControlNodes".sepaClamp.sequence.status.seqActive )
      wire#w1
      I_Contact( "Unit1.Em7.ControlNodes".cmSepaClampTopUpDown.monitoring.inHomePos )
      wire#w2
      Coil( "Unit1.Em7.ControlNodes".sepaClamp."step".action1[220] )
   END_RUNG
   RUNG wire#w1
      I_Contact( "Unit1.Em7.ControlNodes".cmSepaClampBottomUpDown.monitoring.inHomePos )
   END_RUNG wire#w2
   RUNG wire#w1
      Contact( "Unit1.Em7.ControlNodes".cmSepaClampTopUpDown.monitoring.inHomePos )
      Contact( "Unit1.Em7.ControlNodes".cmSepaClampBottomUpDown.monitoring.inHomePos )
      Coil( "Unit1.Em7.ControlNodes".sepaClamp."step".transition1[220] )
   END_RUNG
   RUNG wire#w1
      Contact( "Unit1.Em7.ControlNodes".sepaClamp."step".transition1[220] )
      { S7_Templates := "time_type := Time" } #statTonTime[220].TON(pt := T#100ms, et =>)
      Move(in := #JOB_2_STEP_21, out1 => "Unit1.Em7.ControlNodes".sepaClamp.sequence.status.nextStep)
   END_RUNG
   // the same network as SCL:
   #_w1 := ("Unit1.Em7.ControlNodes".sepaClamp.sequence.status.currentStep = #JOB_2_STEP_20) AND "Unit1.Em7.ControlNodes".sepaClamp.sequence.status.seqActive;
   "Unit1.Em7.ControlNodes".sepaClamp."step".action1[220] := #_w1 AND (NOT "Unit1.Em7.ControlNodes".cmSepaClampTopUpDown.monitoring.inHomePos OR NOT "Unit1.Em7.ControlNodes".cmSepaClampBottomUpDown.monitoring.inHomePos);
   "Unit1.Em7.ControlNodes".sepaClamp."step".transition1[220] := #_w1 AND "Unit1.Em7.ControlNodes".cmSepaClampTopUpDown.monitoring.inHomePos AND "Unit1.Em7.ControlNodes".cmSepaClampBottomUpDown.monitoring.inHomePos;
   #statTonTime[220].TON(IN := #_w1 AND "Unit1.Em7.ControlNodes".sepaClamp."step".transition1[220],
                         PT := T#100ms);
   IF #statTonTime[220].Q THEN
       "Unit1.Em7.ControlNodes".sepaClamp.sequence.status.nextStep := #JOB_2_STEP_21;
   END_IF;
END_REGION

REGION Network 18: Step[221] : Sepa Clamp → Sepa Gripper [Loading Ready]
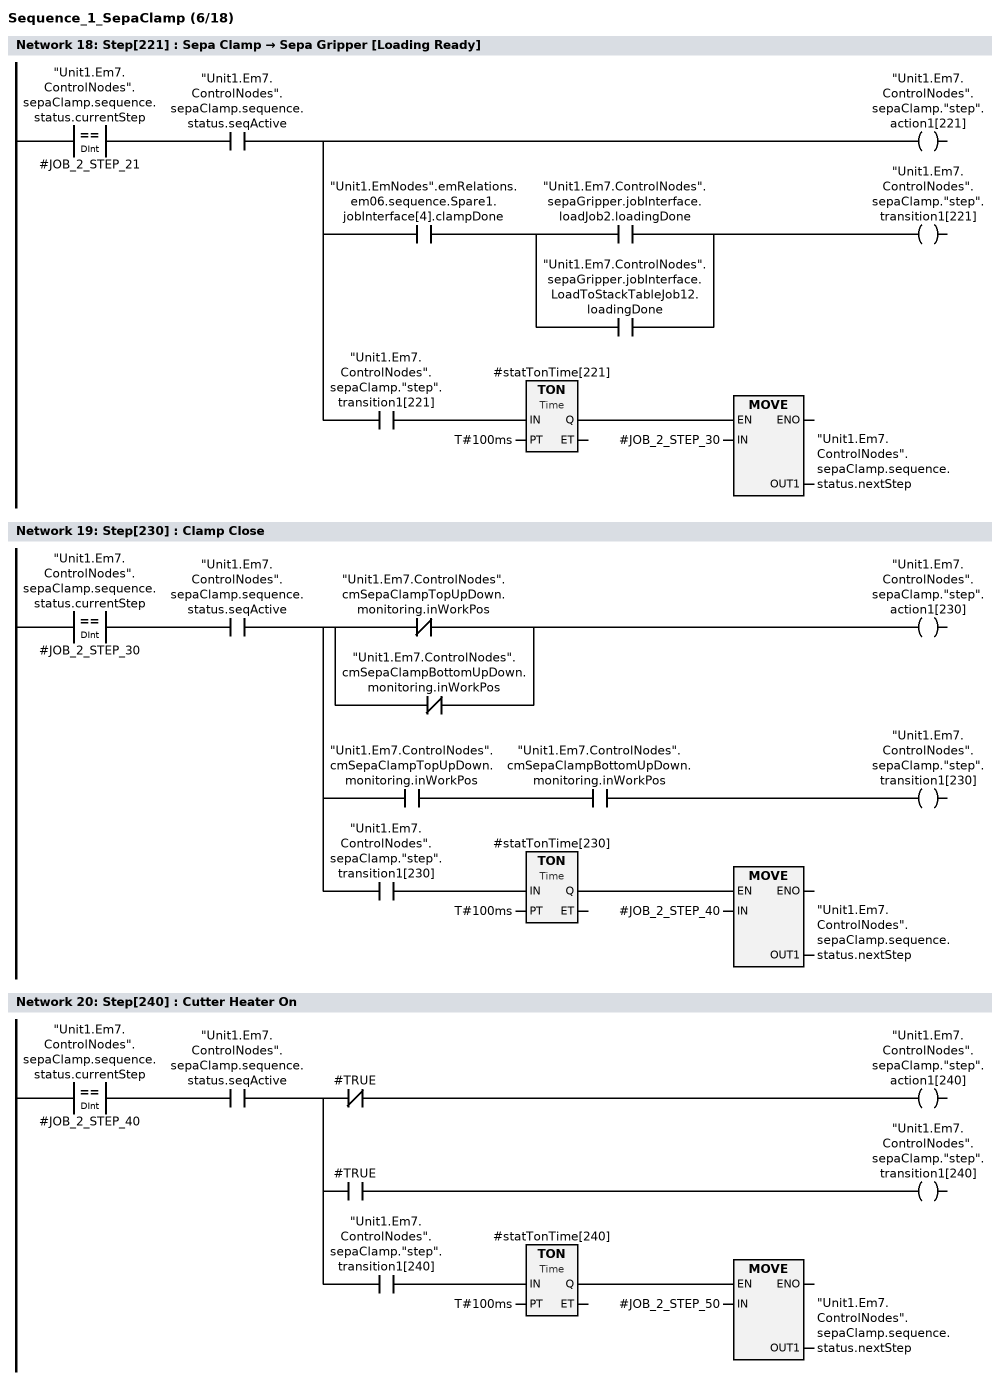
   RUNG wire#powerrail
      { S7_Templates := "SrcType := DInt" } EQ_Contact(in1 := "Unit1.Em7.ControlNodes".sepaClamp.sequence.status.currentStep, in2 := #JOB_2_STEP_21)
      Contact( "Unit1.Em7.ControlNodes".sepaClamp.sequence.status.seqActive )
      wire#w1
      Coil( "Unit1.Em7.ControlNodes".sepaClamp."step".action1[221] )
   END_RUNG
   RUNG wire#w1
      Contact( "Unit1.EmNodes".emRelations.em06.sequence.Spare1.jobInterface[4].clampDone )
      wire#w2
      Contact( "Unit1.Em7.ControlNodes".sepaGripper.jobInterface.loadJob2.loadingDone )
      wire#w3
      Coil( "Unit1.Em7.ControlNodes".sepaClamp."step".transition1[221] )
   END_RUNG
   RUNG wire#w2
      Contact( "Unit1.Em7.ControlNodes".sepaGripper.jobInterface.LoadToStackTableJob12.loadingDone )
   END_RUNG wire#w3
   RUNG wire#w1
      Contact( "Unit1.Em7.ControlNodes".sepaClamp."step".transition1[221] )
      { S7_Templates := "time_type := Time" } #statTonTime[221].TON(pt := T#100ms, et =>)
      Move(in := #JOB_2_STEP_30, out1 => "Unit1.Em7.ControlNodes".sepaClamp.sequence.status.nextStep)
   END_RUNG
   // the same network as SCL:
   "Unit1.Em7.ControlNodes".sepaClamp."step".action1[221] := ("Unit1.Em7.ControlNodes".sepaClamp.sequence.status.currentStep = #JOB_2_STEP_21) AND "Unit1.Em7.ControlNodes".sepaClamp.sequence.status.seqActive;
   "Unit1.Em7.ControlNodes".sepaClamp."step".transition1[221] := ("Unit1.Em7.ControlNodes".sepaClamp.sequence.status.currentStep = #JOB_2_STEP_21) AND "Unit1.Em7.ControlNodes".sepaClamp.sequence.status.seqActive AND "Unit1.EmNodes".emRelations.em06.sequence.Spare1.jobInterface[4].clampDone AND ("Unit1.Em7.ControlNodes".sepaGripper.jobInterface.loadJob2.loadingDone OR "Unit1.Em7.ControlNodes".sepaGripper.jobInterface.LoadToStackTableJob12.loadingDone);
   #statTonTime[221].TON(IN := ("Unit1.Em7.ControlNodes".sepaClamp.sequence.status.currentStep = #JOB_2_STEP_21) AND "Unit1.Em7.ControlNodes".sepaClamp.sequence.status.seqActive AND "Unit1.Em7.ControlNodes".sepaClamp."step".transition1[221],
                         PT := T#100ms);
   IF #statTonTime[221].Q THEN
       "Unit1.Em7.ControlNodes".sepaClamp.sequence.status.nextStep := #JOB_2_STEP_30;
   END_IF;
END_REGION

REGION Network 19: Step[230] : Clamp Close
   RUNG wire#powerrail
      { S7_Templates := "SrcType := DInt" } EQ_Contact(in1 := "Unit1.Em7.ControlNodes".sepaClamp.sequence.status.currentStep, in2 := #JOB_2_STEP_30)
      Contact( "Unit1.Em7.ControlNodes".sepaClamp.sequence.status.seqActive )
      wire#w1
      I_Contact( "Unit1.Em7.ControlNodes".cmSepaClampTopUpDown.monitoring.inWorkPos )
      wire#w2
      Coil( "Unit1.Em7.ControlNodes".sepaClamp."step".action1[230] )
   END_RUNG
   RUNG wire#w1
      I_Contact( "Unit1.Em7.ControlNodes".cmSepaClampBottomUpDown.monitoring.inWorkPos )
   END_RUNG wire#w2
   RUNG wire#w1
      Contact( "Unit1.Em7.ControlNodes".cmSepaClampTopUpDown.monitoring.inWorkPos )
      Contact( "Unit1.Em7.ControlNodes".cmSepaClampBottomUpDown.monitoring.inWorkPos )
      Coil( "Unit1.Em7.ControlNodes".sepaClamp."step".transition1[230] )
   END_RUNG
   RUNG wire#w1
      Contact( "Unit1.Em7.ControlNodes".sepaClamp."step".transition1[230] )
      { S7_Templates := "time_type := Time" } #statTonTime[230].TON(pt := T#100ms, et =>)
      Move(in := #JOB_2_STEP_40, out1 => "Unit1.Em7.ControlNodes".sepaClamp.sequence.status.nextStep)
   END_RUNG
   // the same network as SCL:
   #_w1 := ("Unit1.Em7.ControlNodes".sepaClamp.sequence.status.currentStep = #JOB_2_STEP_30) AND "Unit1.Em7.ControlNodes".sepaClamp.sequence.status.seqActive;
   "Unit1.Em7.ControlNodes".sepaClamp."step".action1[230] := #_w1 AND (NOT "Unit1.Em7.ControlNodes".cmSepaClampTopUpDown.monitoring.inWorkPos OR NOT "Unit1.Em7.ControlNodes".cmSepaClampBottomUpDown.monitoring.inWorkPos);
   "Unit1.Em7.ControlNodes".sepaClamp."step".transition1[230] := #_w1 AND "Unit1.Em7.ControlNodes".cmSepaClampTopUpDown.monitoring.inWorkPos AND "Unit1.Em7.ControlNodes".cmSepaClampBottomUpDown.monitoring.inWorkPos;
   #statTonTime[230].TON(IN := #_w1 AND "Unit1.Em7.ControlNodes".sepaClamp."step".transition1[230],
                         PT := T#100ms);
   IF #statTonTime[230].Q THEN
       "Unit1.Em7.ControlNodes".sepaClamp.sequence.status.nextStep := #JOB_2_STEP_40;
   END_IF;
END_REGION

REGION Network 20: Step[240] : Cutter Heater On
   RUNG wire#powerrail
      { S7_Templates := "SrcType := DInt" } EQ_Contact(in1 := "Unit1.Em7.ControlNodes".sepaClamp.sequence.status.currentStep, in2 := #JOB_2_STEP_40)
      Contact( "Unit1.Em7.ControlNodes".sepaClamp.sequence.status.seqActive )
      wire#w1
      I_Contact( #TRUE )
      Coil( "Unit1.Em7.ControlNodes".sepaClamp."step".action1[240] )
   END_RUNG
   RUNG wire#w1
      Contact( #TRUE )
      Coil( "Unit1.Em7.ControlNodes".sepaClamp."step".transition1[240] )
   END_RUNG
   RUNG wire#w1
      Contact( "Unit1.Em7.ControlNodes".sepaClamp."step".transition1[240] )
      { S7_Templates := "time_type := Time" } #statTonTime[240].TON(pt := T#100ms, et =>)
      Move(in := #JOB_2_STEP_50, out1 => "Unit1.Em7.ControlNodes".sepaClamp.sequence.status.nextStep)
   END_RUNG
   // the same network as SCL:
   #_w1 := ("Unit1.Em7.ControlNodes".sepaClamp.sequence.status.currentStep = #JOB_2_STEP_40) AND "Unit1.Em7.ControlNodes".sepaClamp.sequence.status.seqActive;
   "Unit1.Em7.ControlNodes".sepaClamp."step".action1[240] := #_w1 AND NOT #TRUE;
   "Unit1.Em7.ControlNodes".sepaClamp."step".transition1[240] := #_w1 AND #TRUE;
   #statTonTime[240].TON(IN := #_w1 AND "Unit1.Em7.ControlNodes".sepaClamp."step".transition1[240],
                         PT := T#100ms);
   IF #statTonTime[240].Q THEN
       "Unit1.Em7.ControlNodes".sepaClamp.sequence.status.nextStep := #JOB_2_STEP_50;
   END_IF;
END_REGION

REGION Network 21: Step[250] : Cutter Down
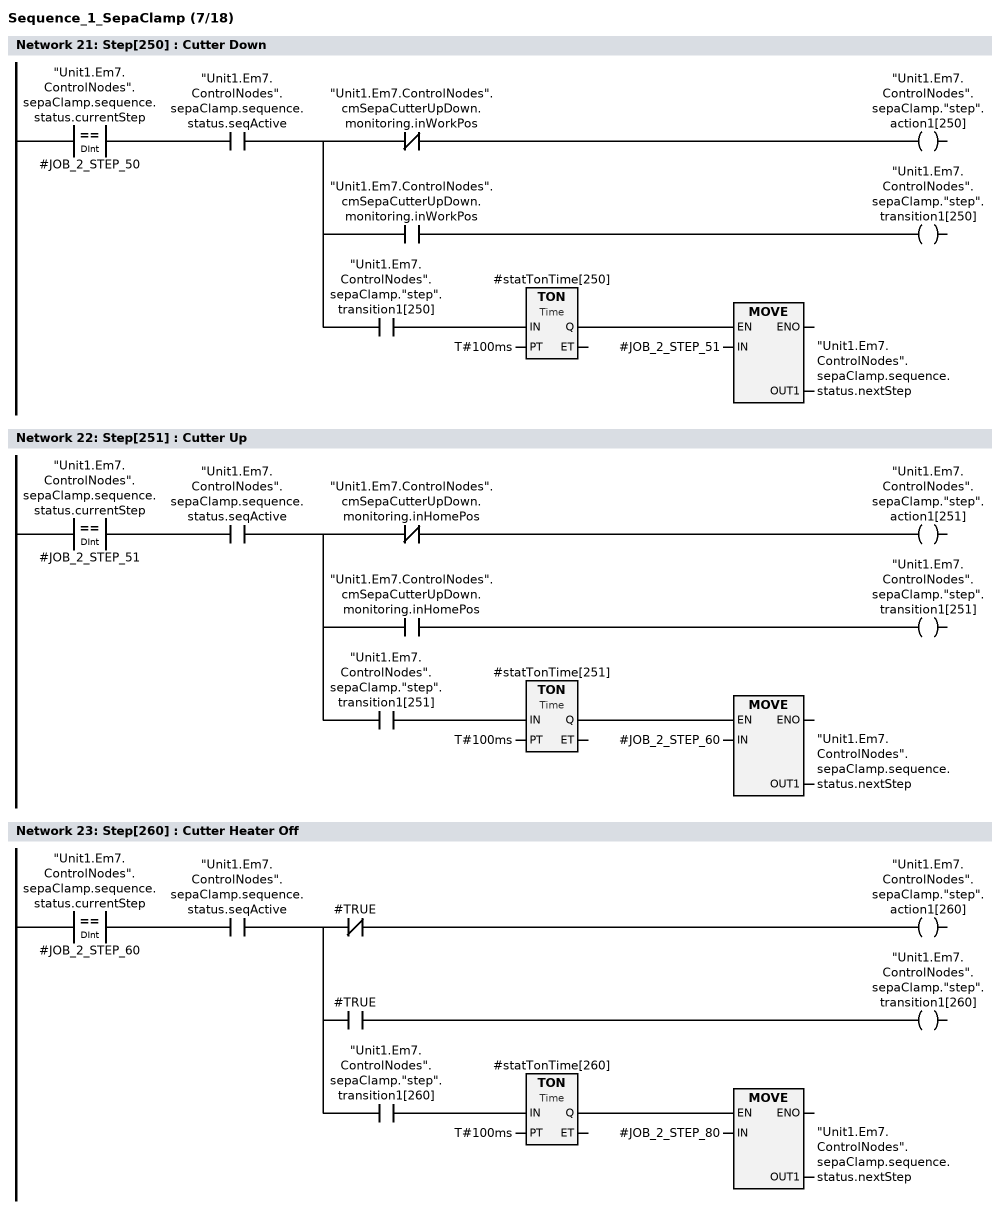
   RUNG wire#powerrail
      { S7_Templates := "SrcType := DInt" } EQ_Contact(in1 := "Unit1.Em7.ControlNodes".sepaClamp.sequence.status.currentStep, in2 := #JOB_2_STEP_50)
      Contact( "Unit1.Em7.ControlNodes".sepaClamp.sequence.status.seqActive )
      wire#w1
      I_Contact( "Unit1.Em7.ControlNodes".cmSepaCutterUpDown.monitoring.inWorkPos )
      Coil( "Unit1.Em7.ControlNodes".sepaClamp."step".action1[250] )
   END_RUNG
   RUNG wire#w1
      Contact( "Unit1.Em7.ControlNodes".cmSepaCutterUpDown.monitoring.inWorkPos )
      Coil( "Unit1.Em7.ControlNodes".sepaClamp."step".transition1[250] )
   END_RUNG
   RUNG wire#w1
      Contact( "Unit1.Em7.ControlNodes".sepaClamp."step".transition1[250] )
      { S7_Templates := "time_type := Time" } #statTonTime[250].TON(pt := T#100ms, et =>)
      Move(in := #JOB_2_STEP_51, out1 => "Unit1.Em7.ControlNodes".sepaClamp.sequence.status.nextStep)
   END_RUNG
   // the same network as SCL:
   #_w1 := ("Unit1.Em7.ControlNodes".sepaClamp.sequence.status.currentStep = #JOB_2_STEP_50) AND "Unit1.Em7.ControlNodes".sepaClamp.sequence.status.seqActive;
   "Unit1.Em7.ControlNodes".sepaClamp."step".action1[250] := #_w1 AND NOT "Unit1.Em7.ControlNodes".cmSepaCutterUpDown.monitoring.inWorkPos;
   "Unit1.Em7.ControlNodes".sepaClamp."step".transition1[250] := #_w1 AND "Unit1.Em7.ControlNodes".cmSepaCutterUpDown.monitoring.inWorkPos;
   #statTonTime[250].TON(IN := #_w1 AND "Unit1.Em7.ControlNodes".sepaClamp."step".transition1[250],
                         PT := T#100ms);
   IF #statTonTime[250].Q THEN
       "Unit1.Em7.ControlNodes".sepaClamp.sequence.status.nextStep := #JOB_2_STEP_51;
   END_IF;
END_REGION

REGION Network 22: Step[251] : Cutter Up
   RUNG wire#powerrail
      { S7_Templates := "SrcType := DInt" } EQ_Contact(in1 := "Unit1.Em7.ControlNodes".sepaClamp.sequence.status.currentStep, in2 := #JOB_2_STEP_51)
      Contact( "Unit1.Em7.ControlNodes".sepaClamp.sequence.status.seqActive )
      wire#w1
      I_Contact( "Unit1.Em7.ControlNodes".cmSepaCutterUpDown.monitoring.inHomePos )
      Coil( "Unit1.Em7.ControlNodes".sepaClamp."step".action1[251] )
   END_RUNG
   RUNG wire#w1
      Contact( "Unit1.Em7.ControlNodes".cmSepaCutterUpDown.monitoring.inHomePos )
      Coil( "Unit1.Em7.ControlNodes".sepaClamp."step".transition1[251] )
   END_RUNG
   RUNG wire#w1
      Contact( "Unit1.Em7.ControlNodes".sepaClamp."step".transition1[251] )
      { S7_Templates := "time_type := Time" } #statTonTime[251].TON(pt := T#100ms, et =>)
      Move(in := #JOB_2_STEP_60, out1 => "Unit1.Em7.ControlNodes".sepaClamp.sequence.status.nextStep)
   END_RUNG
   // the same network as SCL:
   #_w1 := ("Unit1.Em7.ControlNodes".sepaClamp.sequence.status.currentStep = #JOB_2_STEP_51) AND "Unit1.Em7.ControlNodes".sepaClamp.sequence.status.seqActive;
   "Unit1.Em7.ControlNodes".sepaClamp."step".action1[251] := #_w1 AND NOT "Unit1.Em7.ControlNodes".cmSepaCutterUpDown.monitoring.inHomePos;
   "Unit1.Em7.ControlNodes".sepaClamp."step".transition1[251] := #_w1 AND "Unit1.Em7.ControlNodes".cmSepaCutterUpDown.monitoring.inHomePos;
   #statTonTime[251].TON(IN := #_w1 AND "Unit1.Em7.ControlNodes".sepaClamp."step".transition1[251],
                         PT := T#100ms);
   IF #statTonTime[251].Q THEN
       "Unit1.Em7.ControlNodes".sepaClamp.sequence.status.nextStep := #JOB_2_STEP_60;
   END_IF;
END_REGION

REGION Network 23: Step[260] : Cutter Heater Off
   RUNG wire#powerrail
      { S7_Templates := "SrcType := DInt" } EQ_Contact(in1 := "Unit1.Em7.ControlNodes".sepaClamp.sequence.status.currentStep, in2 := #JOB_2_STEP_60)
      Contact( "Unit1.Em7.ControlNodes".sepaClamp.sequence.status.seqActive )
      wire#w1
      I_Contact( #TRUE )
      Coil( "Unit1.Em7.ControlNodes".sepaClamp."step".action1[260] )
   END_RUNG
   RUNG wire#w1
      Contact( #TRUE )
      Coil( "Unit1.Em7.ControlNodes".sepaClamp."step".transition1[260] )
   END_RUNG
   RUNG wire#w1
      Contact( "Unit1.Em7.ControlNodes".sepaClamp."step".transition1[260] )
      { S7_Templates := "time_type := Time" } #statTonTime[260].TON(pt := T#100ms, et =>)
      Move(in := #JOB_2_STEP_80, out1 => "Unit1.Em7.ControlNodes".sepaClamp.sequence.status.nextStep)
   END_RUNG
   // the same network as SCL:
   #_w1 := ("Unit1.Em7.ControlNodes".sepaClamp.sequence.status.currentStep = #JOB_2_STEP_60) AND "Unit1.Em7.ControlNodes".sepaClamp.sequence.status.seqActive;
   "Unit1.Em7.ControlNodes".sepaClamp."step".action1[260] := #_w1 AND NOT #TRUE;
   "Unit1.Em7.ControlNodes".sepaClamp."step".transition1[260] := #_w1 AND #TRUE;
   #statTonTime[260].TON(IN := #_w1 AND "Unit1.Em7.ControlNodes".sepaClamp."step".transition1[260],
                         PT := T#100ms);
   IF #statTonTime[260].Q THEN
       "Unit1.Em7.ControlNodes".sepaClamp.sequence.status.nextStep := #JOB_2_STEP_80;
   END_IF;
END_REGION

REGION Network 24: Step[280] : Clamp X,Z-Axis Winding Ready Pos
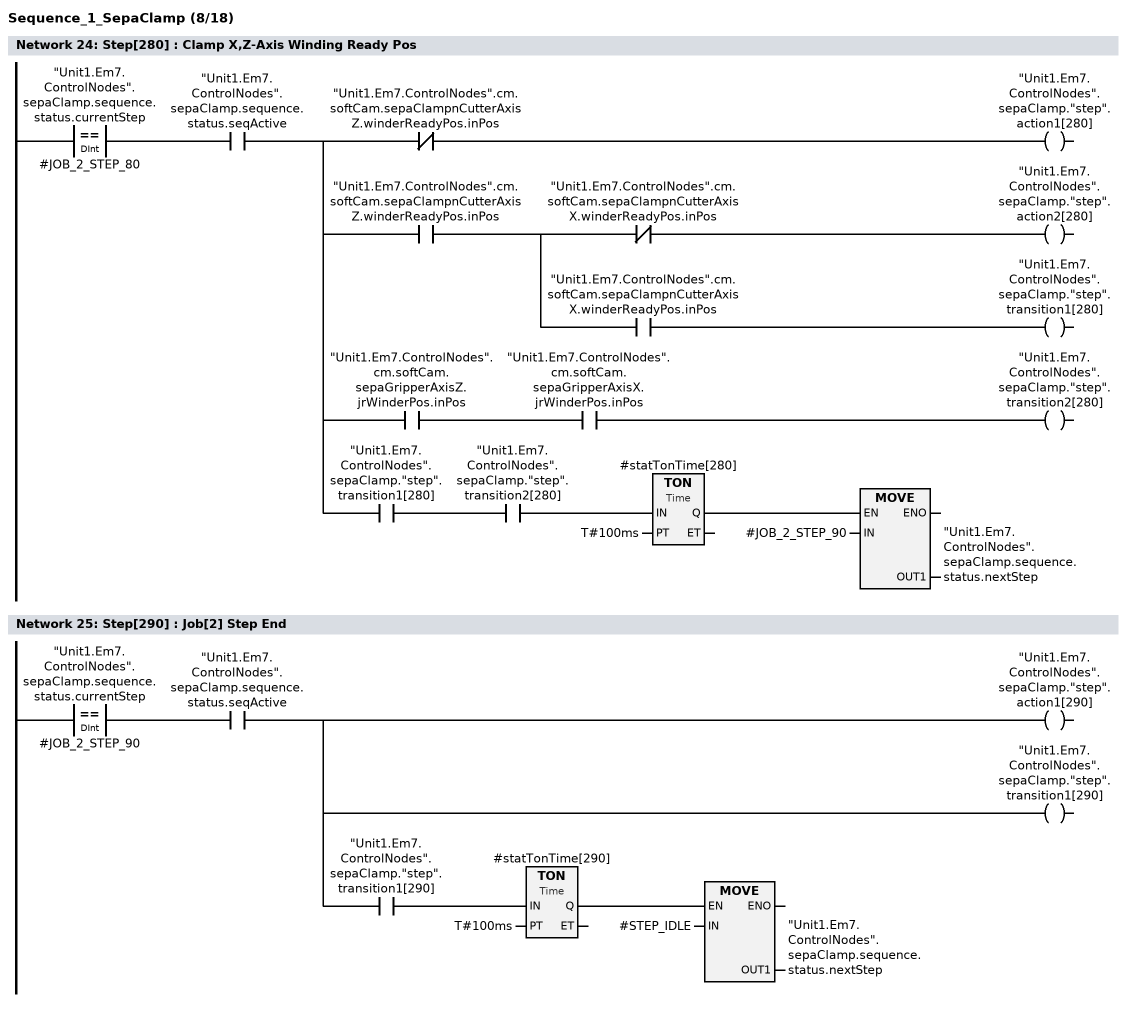
   RUNG wire#powerrail
      { S7_Templates := "SrcType := DInt" } EQ_Contact(in1 := "Unit1.Em7.ControlNodes".sepaClamp.sequence.status.currentStep, in2 := #JOB_2_STEP_80)
      Contact( "Unit1.Em7.ControlNodes".sepaClamp.sequence.status.seqActive )
      wire#w1
      I_Contact( "Unit1.Em7.ControlNodes".cm.softCam.sepaClampnCutterAxisZ.winderReadyPos.inPos )
      Coil( "Unit1.Em7.ControlNodes".sepaClamp."step".action1[280] )
   END_RUNG
   RUNG wire#w1
      Contact( "Unit1.Em7.ControlNodes".cm.softCam.sepaClampnCutterAxisZ.winderReadyPos.inPos )
      wire#w2
      I_Contact( "Unit1.Em7.ControlNodes".cm.softCam.sepaClampnCutterAxisX.winderReadyPos.inPos )
      Coil( "Unit1.Em7.ControlNodes".sepaClamp."step".action2[280] )
   END_RUNG
   RUNG wire#w2
      Contact( "Unit1.Em7.ControlNodes".cm.softCam.sepaClampnCutterAxisX.winderReadyPos.inPos )
      Coil( "Unit1.Em7.ControlNodes".sepaClamp."step".transition1[280] )
   END_RUNG
   RUNG wire#w1
      Contact( "Unit1.Em7.ControlNodes".cm.softCam.sepaGripperAxisZ.jrWinderPos.inPos )
      Contact( "Unit1.Em7.ControlNodes".cm.softCam.sepaGripperAxisX.jrWinderPos.inPos )
      Coil( "Unit1.Em7.ControlNodes".sepaClamp."step".transition2[280] )
   END_RUNG
   RUNG wire#w1
      Contact( "Unit1.Em7.ControlNodes".sepaClamp."step".transition1[280] )
      Contact( "Unit1.Em7.ControlNodes".sepaClamp."step".transition2[280] )
      { S7_Templates := "time_type := Time" } #statTonTime[280].TON(pt := T#100ms, et =>)
      Move(in := #JOB_2_STEP_90, out1 => "Unit1.Em7.ControlNodes".sepaClamp.sequence.status.nextStep)
   END_RUNG
   // the same network as SCL:
   #_w1 := ("Unit1.Em7.ControlNodes".sepaClamp.sequence.status.currentStep = #JOB_2_STEP_80) AND "Unit1.Em7.ControlNodes".sepaClamp.sequence.status.seqActive;
   "Unit1.Em7.ControlNodes".sepaClamp."step".action1[280] := #_w1 AND NOT "Unit1.Em7.ControlNodes".cm.softCam.sepaClampnCutterAxisZ.winderReadyPos.inPos;
   #_w2 := #_w1 AND "Unit1.Em7.ControlNodes".cm.softCam.sepaClampnCutterAxisZ.winderReadyPos.inPos;
   "Unit1.Em7.ControlNodes".sepaClamp."step".action2[280] := #_w2 AND NOT "Unit1.Em7.ControlNodes".cm.softCam.sepaClampnCutterAxisX.winderReadyPos.inPos;
   "Unit1.Em7.ControlNodes".sepaClamp."step".transition1[280] := #_w2 AND "Unit1.Em7.ControlNodes".cm.softCam.sepaClampnCutterAxisX.winderReadyPos.inPos;
   "Unit1.Em7.ControlNodes".sepaClamp."step".transition2[280] := #_w1 AND "Unit1.Em7.ControlNodes".cm.softCam.sepaGripperAxisZ.jrWinderPos.inPos AND "Unit1.Em7.ControlNodes".cm.softCam.sepaGripperAxisX.jrWinderPos.inPos;
   #statTonTime[280].TON(IN := #_w1 AND "Unit1.Em7.ControlNodes".sepaClamp."step".transition1[280] AND "Unit1.Em7.ControlNodes".sepaClamp."step".transition2[280],
                         PT := T#100ms);
   IF #statTonTime[280].Q THEN
       "Unit1.Em7.ControlNodes".sepaClamp.sequence.status.nextStep := #JOB_2_STEP_90;
   END_IF;
END_REGION

REGION Network 25: Step[290] : Job[2] Step End
   RUNG wire#powerrail
      { S7_Templates := "SrcType := DInt" } EQ_Contact(in1 := "Unit1.Em7.ControlNodes".sepaClamp.sequence.status.currentStep, in2 := #JOB_2_STEP_90)
      Contact( "Unit1.Em7.ControlNodes".sepaClamp.sequence.status.seqActive )
      wire#w1
      Coil( "Unit1.Em7.ControlNodes".sepaClamp."step".action1[290] )
   END_RUNG
   RUNG wire#w1
      Coil( "Unit1.Em7.ControlNodes".sepaClamp."step".transition1[290] )
   END_RUNG
   RUNG wire#w1
      Contact( "Unit1.Em7.ControlNodes".sepaClamp."step".transition1[290] )
      { S7_Templates := "time_type := Time" } #statTonTime[290].TON(pt := T#100ms, et =>)
      Move(in := #STEP_IDLE, out1 => "Unit1.Em7.ControlNodes".sepaClamp.sequence.status.nextStep)
   END_RUNG
   // the same network as SCL:
   "Unit1.Em7.ControlNodes".sepaClamp."step".action1[290] := ("Unit1.Em7.ControlNodes".sepaClamp.sequence.status.currentStep = #JOB_2_STEP_90) AND "Unit1.Em7.ControlNodes".sepaClamp.sequence.status.seqActive;
   "Unit1.Em7.ControlNodes".sepaClamp."step".transition1[290] := ("Unit1.Em7.ControlNodes".sepaClamp.sequence.status.currentStep = #JOB_2_STEP_90) AND "Unit1.Em7.ControlNodes".sepaClamp.sequence.status.seqActive;
   #statTonTime[290].TON(IN := ("Unit1.Em7.ControlNodes".sepaClamp.sequence.status.currentStep = #JOB_2_STEP_90) AND "Unit1.Em7.ControlNodes".sepaClamp.sequence.status.seqActive AND "Unit1.Em7.ControlNodes".sepaClamp."step".transition1[290],
                         PT := T#100ms);
   IF #statTonTime[290].Q THEN
       "Unit1.Em7.ControlNodes".sepaClamp.sequence.status.nextStep := #STEP_IDLE;
   END_IF;
END_REGION

REGION Network 26: ******************** JOB[3] Unload ********************
END_REGION

REGION Network 27: Step[301] : JOB[3] Condition
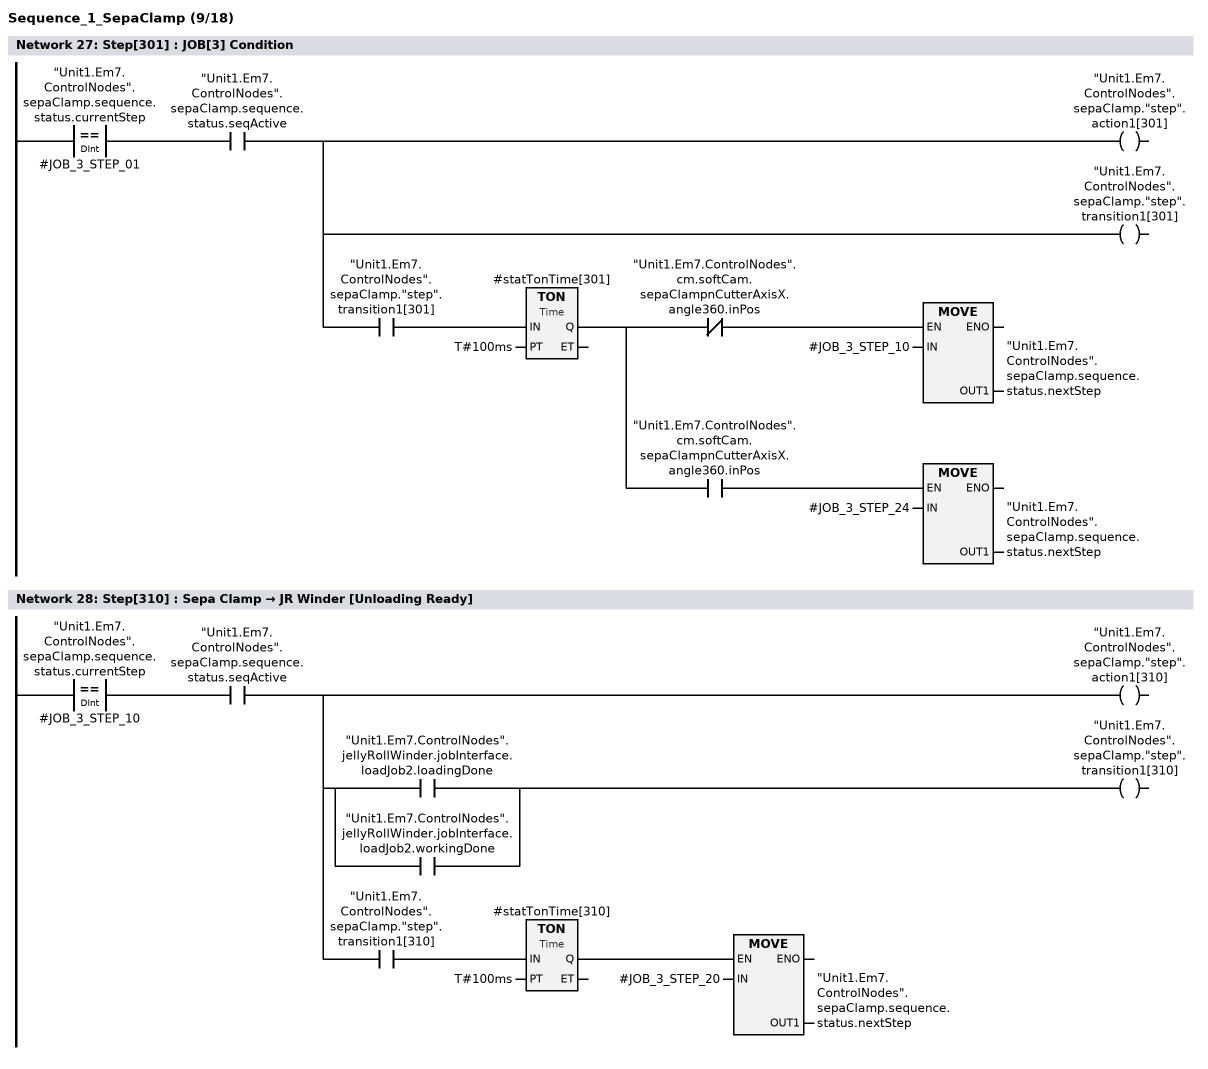
   RUNG wire#powerrail
      { S7_Templates := "SrcType := DInt" } EQ_Contact(in1 := "Unit1.Em7.ControlNodes".sepaClamp.sequence.status.currentStep, in2 := #JOB_3_STEP_01)
      Contact( "Unit1.Em7.ControlNodes".sepaClamp.sequence.status.seqActive )
      wire#w1
      Coil( "Unit1.Em7.ControlNodes".sepaClamp."step".action1[301] )
   END_RUNG
   RUNG wire#w1
      Coil( "Unit1.Em7.ControlNodes".sepaClamp."step".transition1[301] )
   END_RUNG
   RUNG wire#w1
      Contact( "Unit1.Em7.ControlNodes".sepaClamp."step".transition1[301] )
      { S7_Templates := "time_type := Time" } #statTonTime[301].TON(pt := T#100ms, et =>)
      wire#w2
      I_Contact( "Unit1.Em7.ControlNodes".cm.softCam.sepaClampnCutterAxisX.angle360.inPos )
      Move(in := #JOB_3_STEP_10, out1 => "Unit1.Em7.ControlNodes".sepaClamp.sequence.status.nextStep)
   END_RUNG
   RUNG wire#w2
      Contact( "Unit1.Em7.ControlNodes".cm.softCam.sepaClampnCutterAxisX.angle360.inPos )
      Move(in := #JOB_3_STEP_24, out1 => "Unit1.Em7.ControlNodes".sepaClamp.sequence.status.nextStep)
   END_RUNG
   // the same network as SCL:
   "Unit1.Em7.ControlNodes".sepaClamp."step".action1[301] := ("Unit1.Em7.ControlNodes".sepaClamp.sequence.status.currentStep = #JOB_3_STEP_01) AND "Unit1.Em7.ControlNodes".sepaClamp.sequence.status.seqActive;
   "Unit1.Em7.ControlNodes".sepaClamp."step".transition1[301] := ("Unit1.Em7.ControlNodes".sepaClamp.sequence.status.currentStep = #JOB_3_STEP_01) AND "Unit1.Em7.ControlNodes".sepaClamp.sequence.status.seqActive;
   #statTonTime[301].TON(IN := ("Unit1.Em7.ControlNodes".sepaClamp.sequence.status.currentStep = #JOB_3_STEP_01) AND "Unit1.Em7.ControlNodes".sepaClamp.sequence.status.seqActive AND "Unit1.Em7.ControlNodes".sepaClamp."step".transition1[301],
                         PT := T#100ms);
   IF #statTonTime[301].Q AND NOT "Unit1.Em7.ControlNodes".cm.softCam.sepaClampnCutterAxisX.angle360.inPos THEN
       "Unit1.Em7.ControlNodes".sepaClamp.sequence.status.nextStep := #JOB_3_STEP_10;
   END_IF;
   IF #statTonTime[301].Q AND "Unit1.Em7.ControlNodes".cm.softCam.sepaClampnCutterAxisX.angle360.inPos THEN
       "Unit1.Em7.ControlNodes".sepaClamp.sequence.status.nextStep := #JOB_3_STEP_24;
   END_IF;
END_REGION

REGION Network 28: Step[310] : Sepa Clamp → JR Winder [Unloading Ready]
   RUNG wire#powerrail
      { S7_Templates := "SrcType := DInt" } EQ_Contact(in1 := "Unit1.Em7.ControlNodes".sepaClamp.sequence.status.currentStep, in2 := #JOB_3_STEP_10)
      Contact( "Unit1.Em7.ControlNodes".sepaClamp.sequence.status.seqActive )
      wire#w1
      Coil( "Unit1.Em7.ControlNodes".sepaClamp."step".action1[310] )
   END_RUNG
   RUNG wire#w1
      Contact( "Unit1.Em7.ControlNodes".jellyRollWinder.jobInterface.loadJob2.loadingDone )
      wire#w2
      Coil( "Unit1.Em7.ControlNodes".sepaClamp."step".transition1[310] )
   END_RUNG
   RUNG wire#w1
      Contact( "Unit1.Em7.ControlNodes".jellyRollWinder.jobInterface.loadJob2.workingDone )
   END_RUNG wire#w2
   RUNG wire#w1
      Contact( "Unit1.Em7.ControlNodes".sepaClamp."step".transition1[310] )
      { S7_Templates := "time_type := Time" } #statTonTime[310].TON(pt := T#100ms, et =>)
      Move(in := #JOB_3_STEP_20, out1 => "Unit1.Em7.ControlNodes".sepaClamp.sequence.status.nextStep)
   END_RUNG
   // the same network as SCL:
   "Unit1.Em7.ControlNodes".sepaClamp."step".action1[310] := ("Unit1.Em7.ControlNodes".sepaClamp.sequence.status.currentStep = #JOB_3_STEP_10) AND "Unit1.Em7.ControlNodes".sepaClamp.sequence.status.seqActive;
   "Unit1.Em7.ControlNodes".sepaClamp."step".transition1[310] := ("Unit1.Em7.ControlNodes".sepaClamp.sequence.status.currentStep = #JOB_3_STEP_10) AND "Unit1.Em7.ControlNodes".sepaClamp.sequence.status.seqActive AND ("Unit1.Em7.ControlNodes".jellyRollWinder.jobInterface.loadJob2.loadingDone OR "Unit1.Em7.ControlNodes".jellyRollWinder.jobInterface.loadJob2.workingDone);
   #statTonTime[310].TON(IN := ("Unit1.Em7.ControlNodes".sepaClamp.sequence.status.currentStep = #JOB_3_STEP_10) AND "Unit1.Em7.ControlNodes".sepaClamp.sequence.status.seqActive AND "Unit1.Em7.ControlNodes".sepaClamp."step".transition1[310],
                         PT := T#100ms);
   IF #statTonTime[310].Q THEN
       "Unit1.Em7.ControlNodes".sepaClamp.sequence.status.nextStep := #JOB_3_STEP_20;
   END_IF;
END_REGION

REGION Network 29: Step[320] : Clamp X,Z-Axis 90 Angle Pos
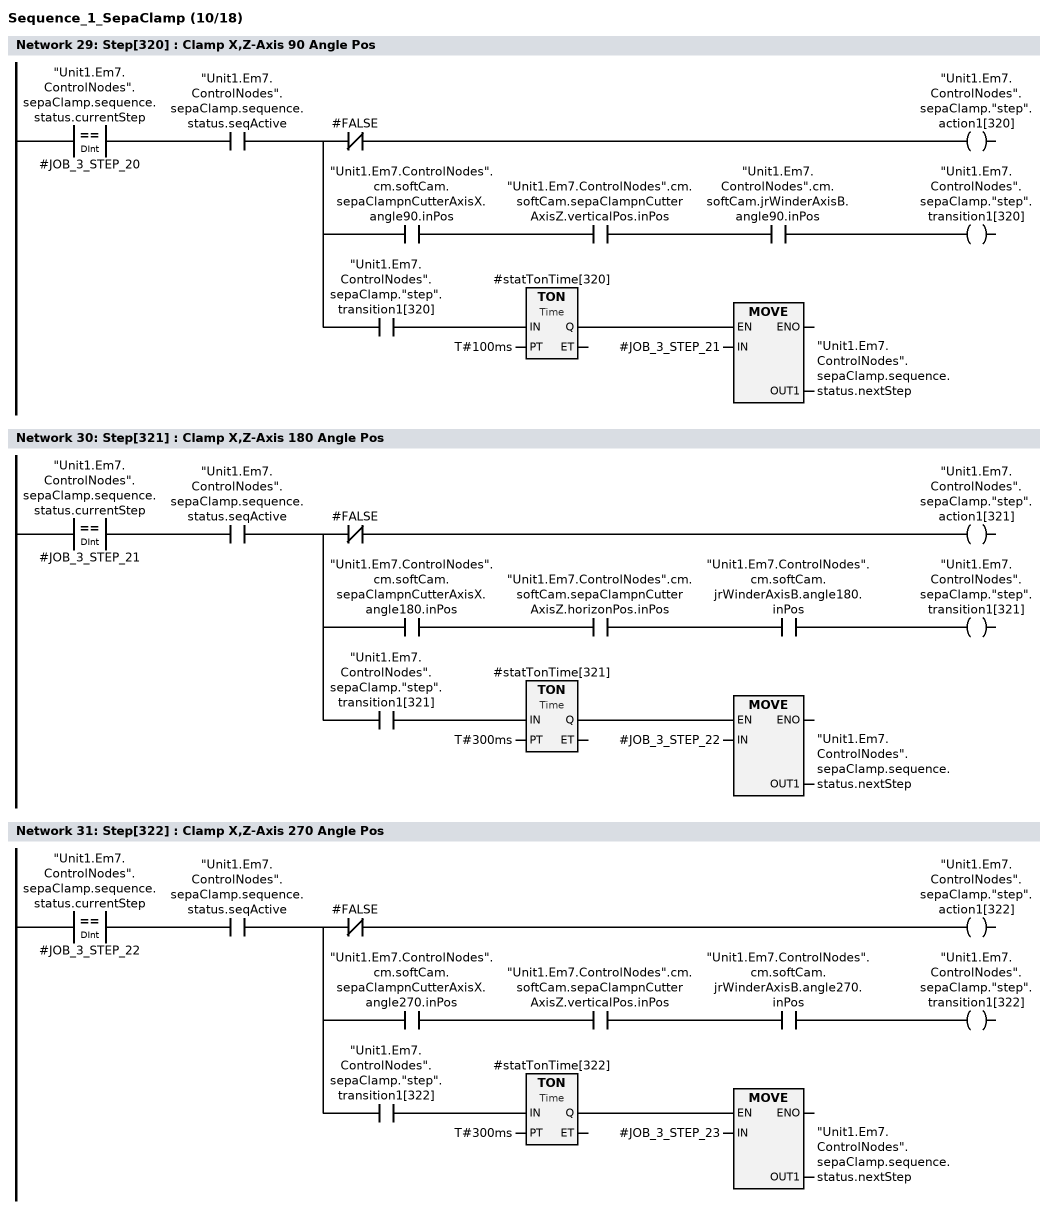
   RUNG wire#powerrail
      { S7_Templates := "SrcType := DInt" } EQ_Contact(in1 := "Unit1.Em7.ControlNodes".sepaClamp.sequence.status.currentStep, in2 := #JOB_3_STEP_20)
      Contact( "Unit1.Em7.ControlNodes".sepaClamp.sequence.status.seqActive )
      wire#w1
      I_Contact( #FALSE )
      Coil( "Unit1.Em7.ControlNodes".sepaClamp."step".action1[320] )
   END_RUNG
   RUNG wire#w1
      Contact( "Unit1.Em7.ControlNodes".cm.softCam.sepaClampnCutterAxisX.angle90.inPos )
      Contact( "Unit1.Em7.ControlNodes".cm.softCam.sepaClampnCutterAxisZ.verticalPos.inPos )
      Contact( "Unit1.Em7.ControlNodes".cm.softCam.jrWinderAxisB.angle90.inPos )
      Coil( "Unit1.Em7.ControlNodes".sepaClamp."step".transition1[320] )
   END_RUNG
   RUNG wire#w1
      Contact( "Unit1.Em7.ControlNodes".sepaClamp."step".transition1[320] )
      { S7_Templates := "time_type := Time" } #statTonTime[320].TON(pt := T#100ms, et =>)
      Move(in := #JOB_3_STEP_21, out1 => "Unit1.Em7.ControlNodes".sepaClamp.sequence.status.nextStep)
   END_RUNG
   // the same network as SCL:
   #_w1 := ("Unit1.Em7.ControlNodes".sepaClamp.sequence.status.currentStep = #JOB_3_STEP_20) AND "Unit1.Em7.ControlNodes".sepaClamp.sequence.status.seqActive;
   "Unit1.Em7.ControlNodes".sepaClamp."step".action1[320] := #_w1 AND NOT #FALSE;
   "Unit1.Em7.ControlNodes".sepaClamp."step".transition1[320] := #_w1 AND "Unit1.Em7.ControlNodes".cm.softCam.sepaClampnCutterAxisX.angle90.inPos AND "Unit1.Em7.ControlNodes".cm.softCam.sepaClampnCutterAxisZ.verticalPos.inPos AND "Unit1.Em7.ControlNodes".cm.softCam.jrWinderAxisB.angle90.inPos;
   #statTonTime[320].TON(IN := #_w1 AND "Unit1.Em7.ControlNodes".sepaClamp."step".transition1[320],
                         PT := T#100ms);
   IF #statTonTime[320].Q THEN
       "Unit1.Em7.ControlNodes".sepaClamp.sequence.status.nextStep := #JOB_3_STEP_21;
   END_IF;
END_REGION

REGION Network 30: Step[321] : Clamp X,Z-Axis 180 Angle Pos
   RUNG wire#powerrail
      { S7_Templates := "SrcType := DInt" } EQ_Contact(in1 := "Unit1.Em7.ControlNodes".sepaClamp.sequence.status.currentStep, in2 := #JOB_3_STEP_21)
      Contact( "Unit1.Em7.ControlNodes".sepaClamp.sequence.status.seqActive )
      wire#w1
      I_Contact( #FALSE )
      Coil( "Unit1.Em7.ControlNodes".sepaClamp."step".action1[321] )
   END_RUNG
   RUNG wire#w1
      Contact( "Unit1.Em7.ControlNodes".cm.softCam.sepaClampnCutterAxisX.angle180.inPos )
      Contact( "Unit1.Em7.ControlNodes".cm.softCam.sepaClampnCutterAxisZ.horizonPos.inPos )
      Contact( "Unit1.Em7.ControlNodes".cm.softCam.jrWinderAxisB.angle180.inPos )
      Coil( "Unit1.Em7.ControlNodes".sepaClamp."step".transition1[321] )
   END_RUNG
   RUNG wire#w1
      Contact( "Unit1.Em7.ControlNodes".sepaClamp."step".transition1[321] )
      { S7_Templates := "time_type := Time" } #statTonTime[321].TON(pt := T#300ms, et =>)
      Move(in := #JOB_3_STEP_22, out1 => "Unit1.Em7.ControlNodes".sepaClamp.sequence.status.nextStep)
   END_RUNG
   // the same network as SCL:
   #_w1 := ("Unit1.Em7.ControlNodes".sepaClamp.sequence.status.currentStep = #JOB_3_STEP_21) AND "Unit1.Em7.ControlNodes".sepaClamp.sequence.status.seqActive;
   "Unit1.Em7.ControlNodes".sepaClamp."step".action1[321] := #_w1 AND NOT #FALSE;
   "Unit1.Em7.ControlNodes".sepaClamp."step".transition1[321] := #_w1 AND "Unit1.Em7.ControlNodes".cm.softCam.sepaClampnCutterAxisX.angle180.inPos AND "Unit1.Em7.ControlNodes".cm.softCam.sepaClampnCutterAxisZ.horizonPos.inPos AND "Unit1.Em7.ControlNodes".cm.softCam.jrWinderAxisB.angle180.inPos;
   #statTonTime[321].TON(IN := #_w1 AND "Unit1.Em7.ControlNodes".sepaClamp."step".transition1[321],
                         PT := T#300ms);
   IF #statTonTime[321].Q THEN
       "Unit1.Em7.ControlNodes".sepaClamp.sequence.status.nextStep := #JOB_3_STEP_22;
   END_IF;
END_REGION

REGION Network 31: Step[322] : Clamp X,Z-Axis 270 Angle Pos
   RUNG wire#powerrail
      { S7_Templates := "SrcType := DInt" } EQ_Contact(in1 := "Unit1.Em7.ControlNodes".sepaClamp.sequence.status.currentStep, in2 := #JOB_3_STEP_22)
      Contact( "Unit1.Em7.ControlNodes".sepaClamp.sequence.status.seqActive )
      wire#w1
      I_Contact( #FALSE )
      Coil( "Unit1.Em7.ControlNodes".sepaClamp."step".action1[322] )
   END_RUNG
   RUNG wire#w1
      Contact( "Unit1.Em7.ControlNodes".cm.softCam.sepaClampnCutterAxisX.angle270.inPos )
      Contact( "Unit1.Em7.ControlNodes".cm.softCam.sepaClampnCutterAxisZ.verticalPos.inPos )
      Contact( "Unit1.Em7.ControlNodes".cm.softCam.jrWinderAxisB.angle270.inPos )
      Coil( "Unit1.Em7.ControlNodes".sepaClamp."step".transition1[322] )
   END_RUNG
   RUNG wire#w1
      Contact( "Unit1.Em7.ControlNodes".sepaClamp."step".transition1[322] )
      { S7_Templates := "time_type := Time" } #statTonTime[322].TON(pt := T#300ms, et =>)
      Move(in := #JOB_3_STEP_23, out1 => "Unit1.Em7.ControlNodes".sepaClamp.sequence.status.nextStep)
   END_RUNG
   // the same network as SCL:
   #_w1 := ("Unit1.Em7.ControlNodes".sepaClamp.sequence.status.currentStep = #JOB_3_STEP_22) AND "Unit1.Em7.ControlNodes".sepaClamp.sequence.status.seqActive;
   "Unit1.Em7.ControlNodes".sepaClamp."step".action1[322] := #_w1 AND NOT #FALSE;
   "Unit1.Em7.ControlNodes".sepaClamp."step".transition1[322] := #_w1 AND "Unit1.Em7.ControlNodes".cm.softCam.sepaClampnCutterAxisX.angle270.inPos AND "Unit1.Em7.ControlNodes".cm.softCam.sepaClampnCutterAxisZ.verticalPos.inPos AND "Unit1.Em7.ControlNodes".cm.softCam.jrWinderAxisB.angle270.inPos;
   #statTonTime[322].TON(IN := #_w1 AND "Unit1.Em7.ControlNodes".sepaClamp."step".transition1[322],
                         PT := T#300ms);
   IF #statTonTime[322].Q THEN
       "Unit1.Em7.ControlNodes".sepaClamp.sequence.status.nextStep := #JOB_3_STEP_23;
   END_IF;
END_REGION

REGION Network 32: Step[323] : Clamp X,Z-Axis 360 Angle Pos
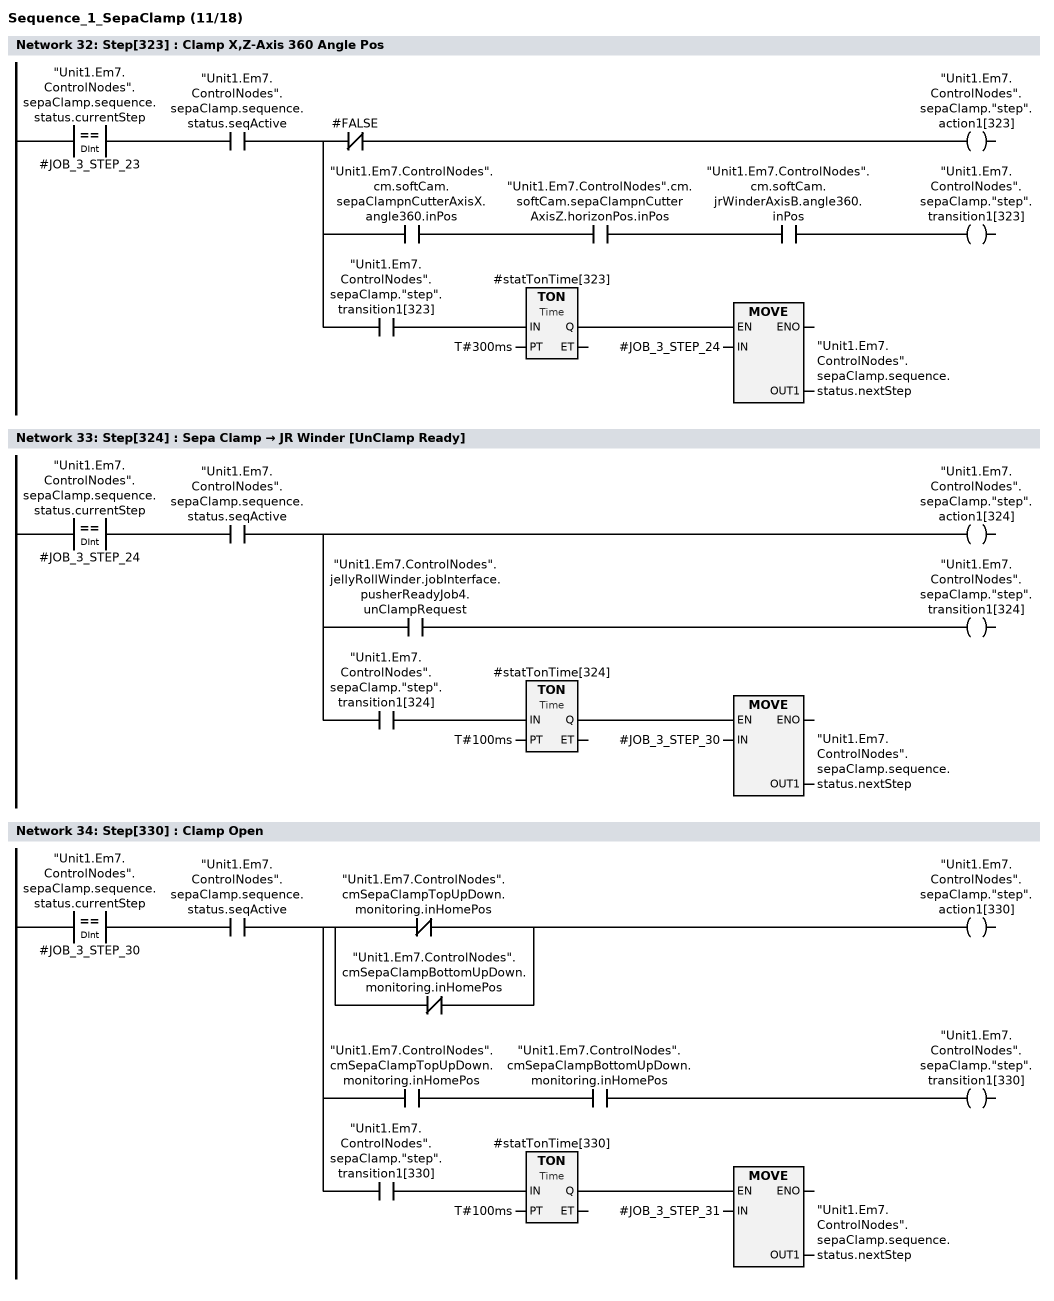
   RUNG wire#powerrail
      { S7_Templates := "SrcType := DInt" } EQ_Contact(in1 := "Unit1.Em7.ControlNodes".sepaClamp.sequence.status.currentStep, in2 := #JOB_3_STEP_23)
      Contact( "Unit1.Em7.ControlNodes".sepaClamp.sequence.status.seqActive )
      wire#w1
      I_Contact( #FALSE )
      Coil( "Unit1.Em7.ControlNodes".sepaClamp."step".action1[323] )
   END_RUNG
   RUNG wire#w1
      Contact( "Unit1.Em7.ControlNodes".cm.softCam.sepaClampnCutterAxisX.angle360.inPos )
      Contact( "Unit1.Em7.ControlNodes".cm.softCam.sepaClampnCutterAxisZ.horizonPos.inPos )
      Contact( "Unit1.Em7.ControlNodes".cm.softCam.jrWinderAxisB.angle360.inPos )
      Coil( "Unit1.Em7.ControlNodes".sepaClamp."step".transition1[323] )
   END_RUNG
   RUNG wire#w1
      Contact( "Unit1.Em7.ControlNodes".sepaClamp."step".transition1[323] )
      { S7_Templates := "time_type := Time" } #statTonTime[323].TON(pt := T#300ms, et =>)
      Move(in := #JOB_3_STEP_24, out1 => "Unit1.Em7.ControlNodes".sepaClamp.sequence.status.nextStep)
   END_RUNG
   // the same network as SCL:
   #_w1 := ("Unit1.Em7.ControlNodes".sepaClamp.sequence.status.currentStep = #JOB_3_STEP_23) AND "Unit1.Em7.ControlNodes".sepaClamp.sequence.status.seqActive;
   "Unit1.Em7.ControlNodes".sepaClamp."step".action1[323] := #_w1 AND NOT #FALSE;
   "Unit1.Em7.ControlNodes".sepaClamp."step".transition1[323] := #_w1 AND "Unit1.Em7.ControlNodes".cm.softCam.sepaClampnCutterAxisX.angle360.inPos AND "Unit1.Em7.ControlNodes".cm.softCam.sepaClampnCutterAxisZ.horizonPos.inPos AND "Unit1.Em7.ControlNodes".cm.softCam.jrWinderAxisB.angle360.inPos;
   #statTonTime[323].TON(IN := #_w1 AND "Unit1.Em7.ControlNodes".sepaClamp."step".transition1[323],
                         PT := T#300ms);
   IF #statTonTime[323].Q THEN
       "Unit1.Em7.ControlNodes".sepaClamp.sequence.status.nextStep := #JOB_3_STEP_24;
   END_IF;
END_REGION

REGION Network 33: Step[324] : Sepa Clamp → JR Winder [UnClamp Ready]
   RUNG wire#powerrail
      { S7_Templates := "SrcType := DInt" } EQ_Contact(in1 := "Unit1.Em7.ControlNodes".sepaClamp.sequence.status.currentStep, in2 := #JOB_3_STEP_24)
      Contact( "Unit1.Em7.ControlNodes".sepaClamp.sequence.status.seqActive )
      wire#w1
      Coil( "Unit1.Em7.ControlNodes".sepaClamp."step".action1[324] )
   END_RUNG
   RUNG wire#w1
      Contact( "Unit1.Em7.ControlNodes".jellyRollWinder.jobInterface.pusherReadyJob4.unClampRequest )
      Coil( "Unit1.Em7.ControlNodes".sepaClamp."step".transition1[324] )
   END_RUNG
   RUNG wire#w1
      Contact( "Unit1.Em7.ControlNodes".sepaClamp."step".transition1[324] )
      { S7_Templates := "time_type := Time" } #statTonTime[324].TON(pt := T#100ms, et =>)
      Move(in := #JOB_3_STEP_30, out1 => "Unit1.Em7.ControlNodes".sepaClamp.sequence.status.nextStep)
   END_RUNG
   // the same network as SCL:
   "Unit1.Em7.ControlNodes".sepaClamp."step".action1[324] := ("Unit1.Em7.ControlNodes".sepaClamp.sequence.status.currentStep = #JOB_3_STEP_24) AND "Unit1.Em7.ControlNodes".sepaClamp.sequence.status.seqActive;
   "Unit1.Em7.ControlNodes".sepaClamp."step".transition1[324] := ("Unit1.Em7.ControlNodes".sepaClamp.sequence.status.currentStep = #JOB_3_STEP_24) AND "Unit1.Em7.ControlNodes".sepaClamp.sequence.status.seqActive AND "Unit1.Em7.ControlNodes".jellyRollWinder.jobInterface.pusherReadyJob4.unClampRequest;
   #statTonTime[324].TON(IN := ("Unit1.Em7.ControlNodes".sepaClamp.sequence.status.currentStep = #JOB_3_STEP_24) AND "Unit1.Em7.ControlNodes".sepaClamp.sequence.status.seqActive AND "Unit1.Em7.ControlNodes".sepaClamp."step".transition1[324],
                         PT := T#100ms);
   IF #statTonTime[324].Q THEN
       "Unit1.Em7.ControlNodes".sepaClamp.sequence.status.nextStep := #JOB_3_STEP_30;
   END_IF;
END_REGION

REGION Network 34: Step[330] : Clamp Open
   RUNG wire#powerrail
      { S7_Templates := "SrcType := DInt" } EQ_Contact(in1 := "Unit1.Em7.ControlNodes".sepaClamp.sequence.status.currentStep, in2 := #JOB_3_STEP_30)
      Contact( "Unit1.Em7.ControlNodes".sepaClamp.sequence.status.seqActive )
      wire#w1
      I_Contact( "Unit1.Em7.ControlNodes".cmSepaClampTopUpDown.monitoring.inHomePos )
      wire#w2
      Coil( "Unit1.Em7.ControlNodes".sepaClamp."step".action1[330] )
   END_RUNG
   RUNG wire#w1
      I_Contact( "Unit1.Em7.ControlNodes".cmSepaClampBottomUpDown.monitoring.inHomePos )
   END_RUNG wire#w2
   RUNG wire#w1
      Contact( "Unit1.Em7.ControlNodes".cmSepaClampTopUpDown.monitoring.inHomePos )
      Contact( "Unit1.Em7.ControlNodes".cmSepaClampBottomUpDown.monitoring.inHomePos )
      Coil( "Unit1.Em7.ControlNodes".sepaClamp."step".transition1[330] )
   END_RUNG
   RUNG wire#w1
      Contact( "Unit1.Em7.ControlNodes".sepaClamp."step".transition1[330] )
      { S7_Templates := "time_type := Time" } #statTonTime[330].TON(pt := T#100ms, et =>)
      Move(in := #JOB_3_STEP_31, out1 => "Unit1.Em7.ControlNodes".sepaClamp.sequence.status.nextStep)
   END_RUNG
   // the same network as SCL:
   #_w1 := ("Unit1.Em7.ControlNodes".sepaClamp.sequence.status.currentStep = #JOB_3_STEP_30) AND "Unit1.Em7.ControlNodes".sepaClamp.sequence.status.seqActive;
   "Unit1.Em7.ControlNodes".sepaClamp."step".action1[330] := #_w1 AND (NOT "Unit1.Em7.ControlNodes".cmSepaClampTopUpDown.monitoring.inHomePos OR NOT "Unit1.Em7.ControlNodes".cmSepaClampBottomUpDown.monitoring.inHomePos);
   "Unit1.Em7.ControlNodes".sepaClamp."step".transition1[330] := #_w1 AND "Unit1.Em7.ControlNodes".cmSepaClampTopUpDown.monitoring.inHomePos AND "Unit1.Em7.ControlNodes".cmSepaClampBottomUpDown.monitoring.inHomePos;
   #statTonTime[330].TON(IN := #_w1 AND "Unit1.Em7.ControlNodes".sepaClamp."step".transition1[330],
                         PT := T#100ms);
   IF #statTonTime[330].Q THEN
       "Unit1.Em7.ControlNodes".sepaClamp.sequence.status.nextStep := #JOB_3_STEP_31;
   END_IF;
END_REGION

REGION Network 35: Step[331] : Sepa Clamp → JR Winder [Unloading Done]
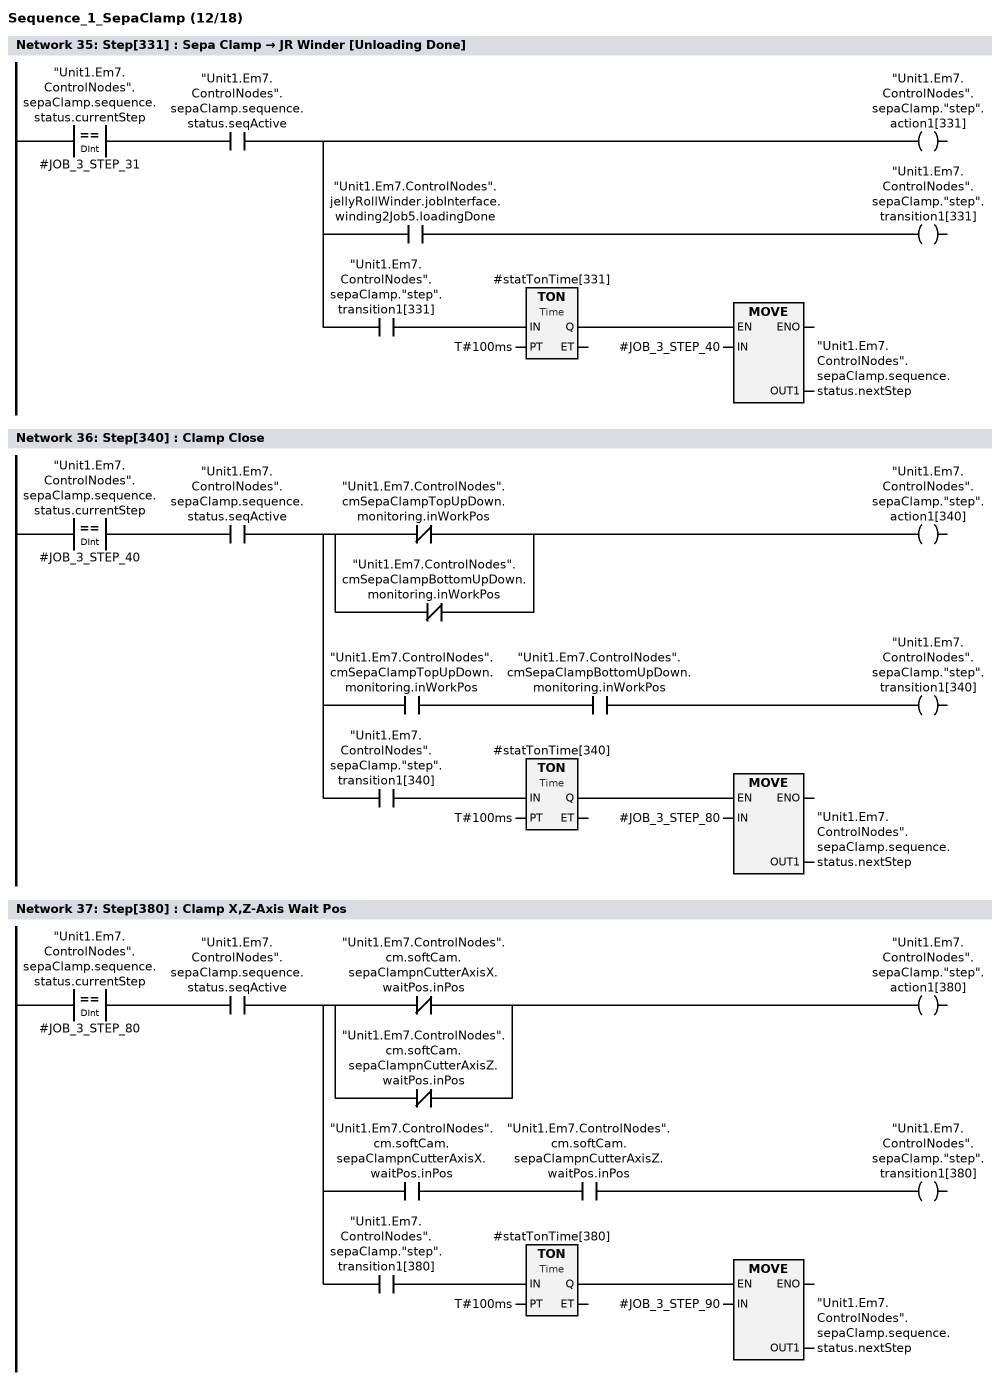
   RUNG wire#powerrail
      { S7_Templates := "SrcType := DInt" } EQ_Contact(in1 := "Unit1.Em7.ControlNodes".sepaClamp.sequence.status.currentStep, in2 := #JOB_3_STEP_31)
      Contact( "Unit1.Em7.ControlNodes".sepaClamp.sequence.status.seqActive )
      wire#w1
      Coil( "Unit1.Em7.ControlNodes".sepaClamp."step".action1[331] )
   END_RUNG
   RUNG wire#w1
      Contact( "Unit1.Em7.ControlNodes".jellyRollWinder.jobInterface.winding2Job5.loadingDone )
      Coil( "Unit1.Em7.ControlNodes".sepaClamp."step".transition1[331] )
   END_RUNG
   RUNG wire#w1
      Contact( "Unit1.Em7.ControlNodes".sepaClamp."step".transition1[331] )
      { S7_Templates := "time_type := Time" } #statTonTime[331].TON(pt := T#100ms, et =>)
      Move(in := #JOB_3_STEP_40, out1 => "Unit1.Em7.ControlNodes".sepaClamp.sequence.status.nextStep)
   END_RUNG
   // the same network as SCL:
   "Unit1.Em7.ControlNodes".sepaClamp."step".action1[331] := ("Unit1.Em7.ControlNodes".sepaClamp.sequence.status.currentStep = #JOB_3_STEP_31) AND "Unit1.Em7.ControlNodes".sepaClamp.sequence.status.seqActive;
   "Unit1.Em7.ControlNodes".sepaClamp."step".transition1[331] := ("Unit1.Em7.ControlNodes".sepaClamp.sequence.status.currentStep = #JOB_3_STEP_31) AND "Unit1.Em7.ControlNodes".sepaClamp.sequence.status.seqActive AND "Unit1.Em7.ControlNodes".jellyRollWinder.jobInterface.winding2Job5.loadingDone;
   #statTonTime[331].TON(IN := ("Unit1.Em7.ControlNodes".sepaClamp.sequence.status.currentStep = #JOB_3_STEP_31) AND "Unit1.Em7.ControlNodes".sepaClamp.sequence.status.seqActive AND "Unit1.Em7.ControlNodes".sepaClamp."step".transition1[331],
                         PT := T#100ms);
   IF #statTonTime[331].Q THEN
       "Unit1.Em7.ControlNodes".sepaClamp.sequence.status.nextStep := #JOB_3_STEP_40;
   END_IF;
END_REGION

REGION Network 36: Step[340] : Clamp Close
   RUNG wire#powerrail
      { S7_Templates := "SrcType := DInt" } EQ_Contact(in1 := "Unit1.Em7.ControlNodes".sepaClamp.sequence.status.currentStep, in2 := #JOB_3_STEP_40)
      Contact( "Unit1.Em7.ControlNodes".sepaClamp.sequence.status.seqActive )
      wire#w1
      I_Contact( "Unit1.Em7.ControlNodes".cmSepaClampTopUpDown.monitoring.inWorkPos )
      wire#w2
      Coil( "Unit1.Em7.ControlNodes".sepaClamp."step".action1[340] )
   END_RUNG
   RUNG wire#w1
      I_Contact( "Unit1.Em7.ControlNodes".cmSepaClampBottomUpDown.monitoring.inWorkPos )
   END_RUNG wire#w2
   RUNG wire#w1
      Contact( "Unit1.Em7.ControlNodes".cmSepaClampTopUpDown.monitoring.inWorkPos )
      Contact( "Unit1.Em7.ControlNodes".cmSepaClampBottomUpDown.monitoring.inWorkPos )
      Coil( "Unit1.Em7.ControlNodes".sepaClamp."step".transition1[340] )
   END_RUNG
   RUNG wire#w1
      Contact( "Unit1.Em7.ControlNodes".sepaClamp."step".transition1[340] )
      { S7_Templates := "time_type := Time" } #statTonTime[340].TON(pt := T#100ms, et =>)
      Move(in := #JOB_3_STEP_80, out1 => "Unit1.Em7.ControlNodes".sepaClamp.sequence.status.nextStep)
   END_RUNG
   // the same network as SCL:
   #_w1 := ("Unit1.Em7.ControlNodes".sepaClamp.sequence.status.currentStep = #JOB_3_STEP_40) AND "Unit1.Em7.ControlNodes".sepaClamp.sequence.status.seqActive;
   "Unit1.Em7.ControlNodes".sepaClamp."step".action1[340] := #_w1 AND (NOT "Unit1.Em7.ControlNodes".cmSepaClampTopUpDown.monitoring.inWorkPos OR NOT "Unit1.Em7.ControlNodes".cmSepaClampBottomUpDown.monitoring.inWorkPos);
   "Unit1.Em7.ControlNodes".sepaClamp."step".transition1[340] := #_w1 AND "Unit1.Em7.ControlNodes".cmSepaClampTopUpDown.monitoring.inWorkPos AND "Unit1.Em7.ControlNodes".cmSepaClampBottomUpDown.monitoring.inWorkPos;
   #statTonTime[340].TON(IN := #_w1 AND "Unit1.Em7.ControlNodes".sepaClamp."step".transition1[340],
                         PT := T#100ms);
   IF #statTonTime[340].Q THEN
       "Unit1.Em7.ControlNodes".sepaClamp.sequence.status.nextStep := #JOB_3_STEP_80;
   END_IF;
END_REGION

REGION Network 37: Step[380] : Clamp X,Z-Axis Wait Pos
   RUNG wire#powerrail
      { S7_Templates := "SrcType := DInt" } EQ_Contact(in1 := "Unit1.Em7.ControlNodes".sepaClamp.sequence.status.currentStep, in2 := #JOB_3_STEP_80)
      Contact( "Unit1.Em7.ControlNodes".sepaClamp.sequence.status.seqActive )
      wire#w1
      I_Contact( "Unit1.Em7.ControlNodes".cm.softCam.sepaClampnCutterAxisX.waitPos.inPos )
      wire#w2
      Coil( "Unit1.Em7.ControlNodes".sepaClamp."step".action1[380] )
   END_RUNG
   RUNG wire#w1
      I_Contact( "Unit1.Em7.ControlNodes".cm.softCam.sepaClampnCutterAxisZ.waitPos.inPos )
   END_RUNG wire#w2
   RUNG wire#w1
      Contact( "Unit1.Em7.ControlNodes".cm.softCam.sepaClampnCutterAxisX.waitPos.inPos )
      Contact( "Unit1.Em7.ControlNodes".cm.softCam.sepaClampnCutterAxisZ.waitPos.inPos )
      Coil( "Unit1.Em7.ControlNodes".sepaClamp."step".transition1[380] )
   END_RUNG
   RUNG wire#w1
      Contact( "Unit1.Em7.ControlNodes".sepaClamp."step".transition1[380] )
      { S7_Templates := "time_type := Time" } #statTonTime[380].TON(pt := T#100ms, et =>)
      Move(in := #JOB_3_STEP_90, out1 => "Unit1.Em7.ControlNodes".sepaClamp.sequence.status.nextStep)
   END_RUNG
   // the same network as SCL:
   #_w1 := ("Unit1.Em7.ControlNodes".sepaClamp.sequence.status.currentStep = #JOB_3_STEP_80) AND "Unit1.Em7.ControlNodes".sepaClamp.sequence.status.seqActive;
   "Unit1.Em7.ControlNodes".sepaClamp."step".action1[380] := #_w1 AND (NOT "Unit1.Em7.ControlNodes".cm.softCam.sepaClampnCutterAxisX.waitPos.inPos OR NOT "Unit1.Em7.ControlNodes".cm.softCam.sepaClampnCutterAxisZ.waitPos.inPos);
   "Unit1.Em7.ControlNodes".sepaClamp."step".transition1[380] := #_w1 AND "Unit1.Em7.ControlNodes".cm.softCam.sepaClampnCutterAxisX.waitPos.inPos AND "Unit1.Em7.ControlNodes".cm.softCam.sepaClampnCutterAxisZ.waitPos.inPos;
   #statTonTime[380].TON(IN := #_w1 AND "Unit1.Em7.ControlNodes".sepaClamp."step".transition1[380],
                         PT := T#100ms);
   IF #statTonTime[380].Q THEN
       "Unit1.Em7.ControlNodes".sepaClamp.sequence.status.nextStep := #JOB_3_STEP_90;
   END_IF;
END_REGION

REGION Network 38: Step[390] : Job[3] Step End
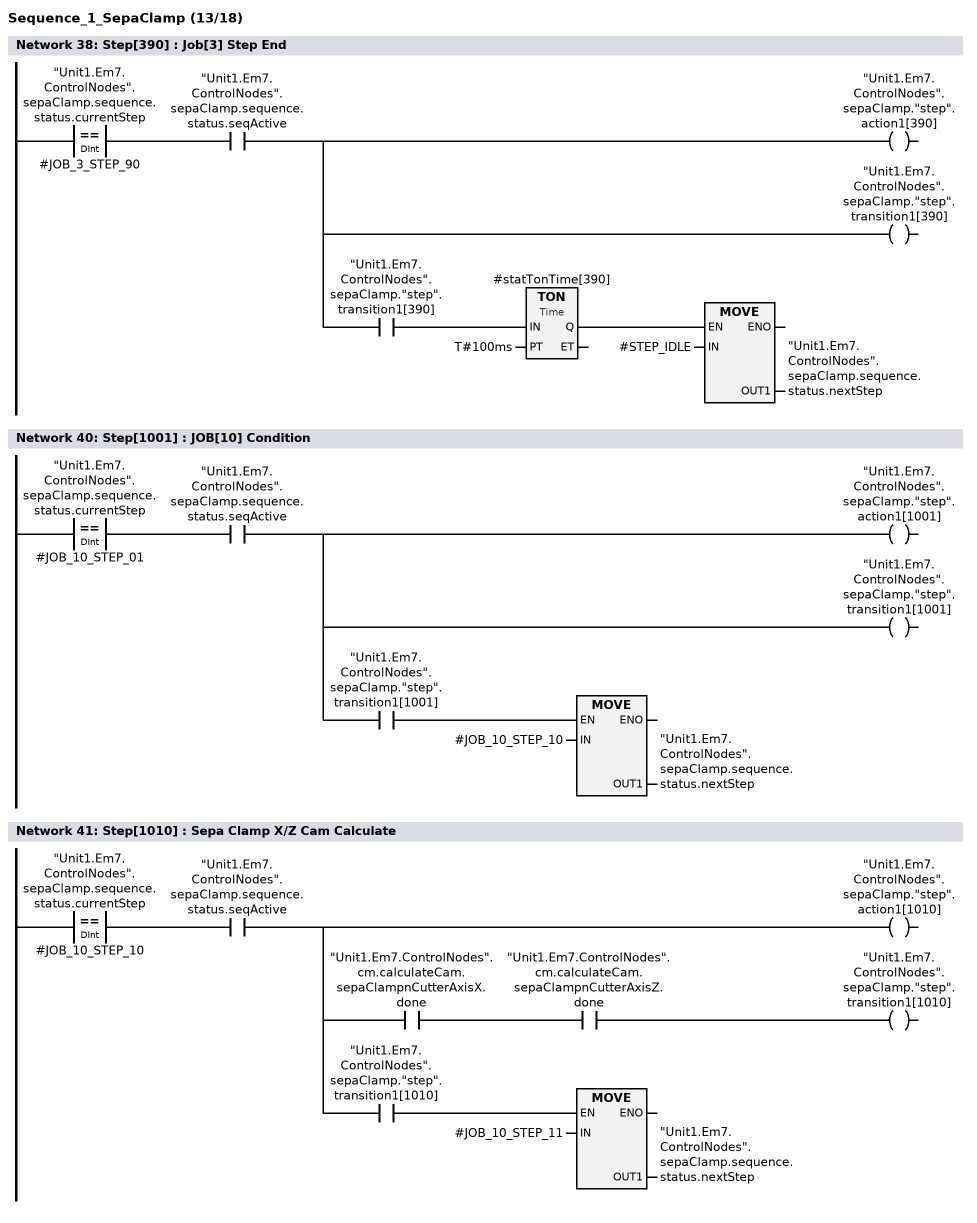
   RUNG wire#powerrail
      { S7_Templates := "SrcType := DInt" } EQ_Contact(in1 := "Unit1.Em7.ControlNodes".sepaClamp.sequence.status.currentStep, in2 := #JOB_3_STEP_90)
      Contact( "Unit1.Em7.ControlNodes".sepaClamp.sequence.status.seqActive )
      wire#w1
      Coil( "Unit1.Em7.ControlNodes".sepaClamp."step".action1[390] )
   END_RUNG
   RUNG wire#w1
      Coil( "Unit1.Em7.ControlNodes".sepaClamp."step".transition1[390] )
   END_RUNG
   RUNG wire#w1
      Contact( "Unit1.Em7.ControlNodes".sepaClamp."step".transition1[390] )
      { S7_Templates := "time_type := Time" } #statTonTime[390].TON(pt := T#100ms, et =>)
      Move(in := #STEP_IDLE, out1 => "Unit1.Em7.ControlNodes".sepaClamp.sequence.status.nextStep)
   END_RUNG
   // the same network as SCL:
   "Unit1.Em7.ControlNodes".sepaClamp."step".action1[390] := ("Unit1.Em7.ControlNodes".sepaClamp.sequence.status.currentStep = #JOB_3_STEP_90) AND "Unit1.Em7.ControlNodes".sepaClamp.sequence.status.seqActive;
   "Unit1.Em7.ControlNodes".sepaClamp."step".transition1[390] := ("Unit1.Em7.ControlNodes".sepaClamp.sequence.status.currentStep = #JOB_3_STEP_90) AND "Unit1.Em7.ControlNodes".sepaClamp.sequence.status.seqActive;
   #statTonTime[390].TON(IN := ("Unit1.Em7.ControlNodes".sepaClamp.sequence.status.currentStep = #JOB_3_STEP_90) AND "Unit1.Em7.ControlNodes".sepaClamp.sequence.status.seqActive AND "Unit1.Em7.ControlNodes".sepaClamp."step".transition1[390],
                         PT := T#100ms);
   IF #statTonTime[390].Q THEN
       "Unit1.Em7.ControlNodes".sepaClamp.sequence.status.nextStep := #STEP_IDLE;
   END_IF;
END_REGION

REGION Network 39: ******************** JOB[10] Unload Cam ********************
END_REGION

REGION Network 40: Step[1001] : JOB[10] Condition
   RUNG wire#powerrail
      { S7_Templates := "SrcType := DInt" } EQ_Contact(in1 := "Unit1.Em7.ControlNodes".sepaClamp.sequence.status.currentStep, in2 := #JOB_10_STEP_01)
      Contact( "Unit1.Em7.ControlNodes".sepaClamp.sequence.status.seqActive )
      wire#w1
      Coil( "Unit1.Em7.ControlNodes".sepaClamp."step".action1[1001] )
   END_RUNG
   RUNG wire#w1
      Coil( "Unit1.Em7.ControlNodes".sepaClamp."step".transition1[1001] )
   END_RUNG
   RUNG wire#w1
      Contact( "Unit1.Em7.ControlNodes".sepaClamp."step".transition1[1001] )
      Move(in := #JOB_10_STEP_10, out1 => "Unit1.Em7.ControlNodes".sepaClamp.sequence.status.nextStep)
   END_RUNG
   // the same network as SCL:
   "Unit1.Em7.ControlNodes".sepaClamp."step".action1[1001] := ("Unit1.Em7.ControlNodes".sepaClamp.sequence.status.currentStep = #JOB_10_STEP_01) AND "Unit1.Em7.ControlNodes".sepaClamp.sequence.status.seqActive;
   "Unit1.Em7.ControlNodes".sepaClamp."step".transition1[1001] := ("Unit1.Em7.ControlNodes".sepaClamp.sequence.status.currentStep = #JOB_10_STEP_01) AND "Unit1.Em7.ControlNodes".sepaClamp.sequence.status.seqActive;
   IF ("Unit1.Em7.ControlNodes".sepaClamp.sequence.status.currentStep = #JOB_10_STEP_01) AND "Unit1.Em7.ControlNodes".sepaClamp.sequence.status.seqActive AND "Unit1.Em7.ControlNodes".sepaClamp."step".transition1[1001] THEN
       "Unit1.Em7.ControlNodes".sepaClamp.sequence.status.nextStep := #JOB_10_STEP_10;
   END_IF;
END_REGION

REGION Network 41: Step[1010] : Sepa Clamp X/Z Cam Calculate
   RUNG wire#powerrail
      { S7_Templates := "SrcType := DInt" } EQ_Contact(in1 := "Unit1.Em7.ControlNodes".sepaClamp.sequence.status.currentStep, in2 := #JOB_10_STEP_10)
      Contact( "Unit1.Em7.ControlNodes".sepaClamp.sequence.status.seqActive )
      wire#w1
      Coil( "Unit1.Em7.ControlNodes".sepaClamp."step".action1[1010] )
   END_RUNG
   RUNG wire#w1
      Contact( "Unit1.Em7.ControlNodes".cm.calculateCam.sepaClampnCutterAxisX.done )
      Contact( "Unit1.Em7.ControlNodes".cm.calculateCam.sepaClampnCutterAxisZ.done )
      Coil( "Unit1.Em7.ControlNodes".sepaClamp."step".transition1[1010] )
   END_RUNG
   RUNG wire#w1
      Contact( "Unit1.Em7.ControlNodes".sepaClamp."step".transition1[1010] )
      Move(in := #JOB_10_STEP_11, out1 => "Unit1.Em7.ControlNodes".sepaClamp.sequence.status.nextStep)
   END_RUNG
   // the same network as SCL:
   "Unit1.Em7.ControlNodes".sepaClamp."step".action1[1010] := ("Unit1.Em7.ControlNodes".sepaClamp.sequence.status.currentStep = #JOB_10_STEP_10) AND "Unit1.Em7.ControlNodes".sepaClamp.sequence.status.seqActive;
   "Unit1.Em7.ControlNodes".sepaClamp."step".transition1[1010] := ("Unit1.Em7.ControlNodes".sepaClamp.sequence.status.currentStep = #JOB_10_STEP_10) AND "Unit1.Em7.ControlNodes".sepaClamp.sequence.status.seqActive AND "Unit1.Em7.ControlNodes".cm.calculateCam.sepaClampnCutterAxisX.done AND "Unit1.Em7.ControlNodes".cm.calculateCam.sepaClampnCutterAxisZ.done;
   IF ("Unit1.Em7.ControlNodes".sepaClamp.sequence.status.currentStep = #JOB_10_STEP_10) AND "Unit1.Em7.ControlNodes".sepaClamp.sequence.status.seqActive AND "Unit1.Em7.ControlNodes".sepaClamp."step".transition1[1010] THEN
       "Unit1.Em7.ControlNodes".sepaClamp.sequence.status.nextStep := #JOB_10_STEP_11;
   END_IF;
END_REGION

REGION Network 42: Step[1011] : Sepa Clamp X/Z CamIn [InSync]
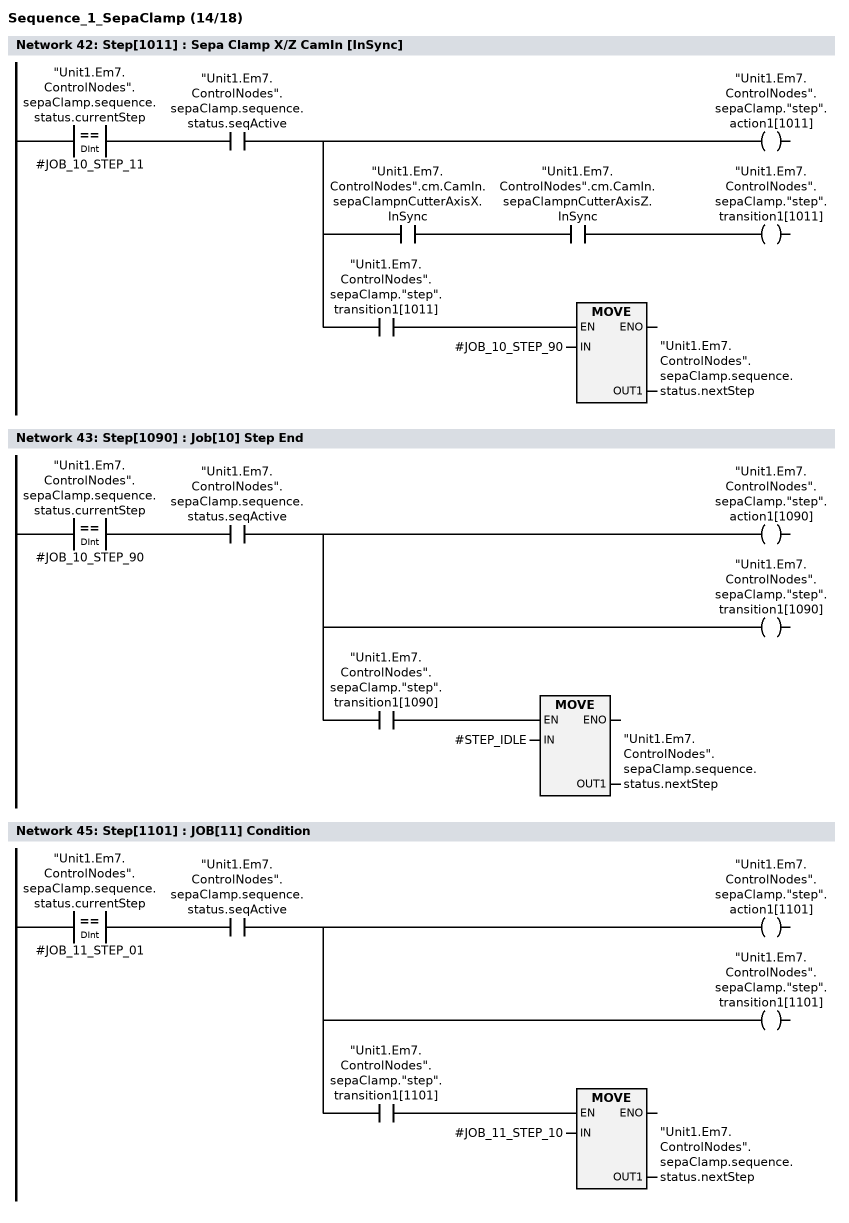
   RUNG wire#powerrail
      { S7_Templates := "SrcType := DInt" } EQ_Contact(in1 := "Unit1.Em7.ControlNodes".sepaClamp.sequence.status.currentStep, in2 := #JOB_10_STEP_11)
      Contact( "Unit1.Em7.ControlNodes".sepaClamp.sequence.status.seqActive )
      wire#w1
      Coil( "Unit1.Em7.ControlNodes".sepaClamp."step".action1[1011] )
   END_RUNG
   RUNG wire#w1
      Contact( "Unit1.Em7.ControlNodes".cm.CamIn.sepaClampnCutterAxisX.InSync )
      Contact( "Unit1.Em7.ControlNodes".cm.CamIn.sepaClampnCutterAxisZ.InSync )
      Coil( "Unit1.Em7.ControlNodes".sepaClamp."step".transition1[1011] )
   END_RUNG
   RUNG wire#w1
      Contact( "Unit1.Em7.ControlNodes".sepaClamp."step".transition1[1011] )
      Move(in := #JOB_10_STEP_90, out1 => "Unit1.Em7.ControlNodes".sepaClamp.sequence.status.nextStep)
   END_RUNG
   // the same network as SCL:
   "Unit1.Em7.ControlNodes".sepaClamp."step".action1[1011] := ("Unit1.Em7.ControlNodes".sepaClamp.sequence.status.currentStep = #JOB_10_STEP_11) AND "Unit1.Em7.ControlNodes".sepaClamp.sequence.status.seqActive;
   "Unit1.Em7.ControlNodes".sepaClamp."step".transition1[1011] := ("Unit1.Em7.ControlNodes".sepaClamp.sequence.status.currentStep = #JOB_10_STEP_11) AND "Unit1.Em7.ControlNodes".sepaClamp.sequence.status.seqActive AND "Unit1.Em7.ControlNodes".cm.CamIn.sepaClampnCutterAxisX.InSync AND "Unit1.Em7.ControlNodes".cm.CamIn.sepaClampnCutterAxisZ.InSync;
   IF ("Unit1.Em7.ControlNodes".sepaClamp.sequence.status.currentStep = #JOB_10_STEP_11) AND "Unit1.Em7.ControlNodes".sepaClamp.sequence.status.seqActive AND "Unit1.Em7.ControlNodes".sepaClamp."step".transition1[1011] THEN
       "Unit1.Em7.ControlNodes".sepaClamp.sequence.status.nextStep := #JOB_10_STEP_90;
   END_IF;
END_REGION

REGION Network 43: Step[1090] : Job[10] Step End
   RUNG wire#powerrail
      { S7_Templates := "SrcType := DInt" } EQ_Contact(in1 := "Unit1.Em7.ControlNodes".sepaClamp.sequence.status.currentStep, in2 := #JOB_10_STEP_90)
      Contact( "Unit1.Em7.ControlNodes".sepaClamp.sequence.status.seqActive )
      wire#w1
      Coil( "Unit1.Em7.ControlNodes".sepaClamp."step".action1[1090] )
   END_RUNG
   RUNG wire#w1
      Coil( "Unit1.Em7.ControlNodes".sepaClamp."step".transition1[1090] )
   END_RUNG
   RUNG wire#w1
      Contact( "Unit1.Em7.ControlNodes".sepaClamp."step".transition1[1090] )
      Move(in := #STEP_IDLE, out1 => "Unit1.Em7.ControlNodes".sepaClamp.sequence.status.nextStep)
   END_RUNG
   // the same network as SCL:
   "Unit1.Em7.ControlNodes".sepaClamp."step".action1[1090] := ("Unit1.Em7.ControlNodes".sepaClamp.sequence.status.currentStep = #JOB_10_STEP_90) AND "Unit1.Em7.ControlNodes".sepaClamp.sequence.status.seqActive;
   "Unit1.Em7.ControlNodes".sepaClamp."step".transition1[1090] := ("Unit1.Em7.ControlNodes".sepaClamp.sequence.status.currentStep = #JOB_10_STEP_90) AND "Unit1.Em7.ControlNodes".sepaClamp.sequence.status.seqActive;
   IF ("Unit1.Em7.ControlNodes".sepaClamp.sequence.status.currentStep = #JOB_10_STEP_90) AND "Unit1.Em7.ControlNodes".sepaClamp.sequence.status.seqActive AND "Unit1.Em7.ControlNodes".sepaClamp."step".transition1[1090] THEN
       "Unit1.Em7.ControlNodes".sepaClamp.sequence.status.nextStep := #STEP_IDLE;
   END_IF;
END_REGION

REGION Network 44: ******************** JOB[11] Unload Stop Sync ********************
END_REGION

REGION Network 45: Step[1101] : JOB[11] Condition
   RUNG wire#powerrail
      { S7_Templates := "SrcType := DInt" } EQ_Contact(in1 := "Unit1.Em7.ControlNodes".sepaClamp.sequence.status.currentStep, in2 := #JOB_11_STEP_01)
      Contact( "Unit1.Em7.ControlNodes".sepaClamp.sequence.status.seqActive )
      wire#w1
      Coil( "Unit1.Em7.ControlNodes".sepaClamp."step".action1[1101] )
   END_RUNG
   RUNG wire#w1
      Coil( "Unit1.Em7.ControlNodes".sepaClamp."step".transition1[1101] )
   END_RUNG
   RUNG wire#w1
      Contact( "Unit1.Em7.ControlNodes".sepaClamp."step".transition1[1101] )
      Move(in := #JOB_11_STEP_10, out1 => "Unit1.Em7.ControlNodes".sepaClamp.sequence.status.nextStep)
   END_RUNG
   // the same network as SCL:
   "Unit1.Em7.ControlNodes".sepaClamp."step".action1[1101] := ("Unit1.Em7.ControlNodes".sepaClamp.sequence.status.currentStep = #JOB_11_STEP_01) AND "Unit1.Em7.ControlNodes".sepaClamp.sequence.status.seqActive;
   "Unit1.Em7.ControlNodes".sepaClamp."step".transition1[1101] := ("Unit1.Em7.ControlNodes".sepaClamp.sequence.status.currentStep = #JOB_11_STEP_01) AND "Unit1.Em7.ControlNodes".sepaClamp.sequence.status.seqActive;
   IF ("Unit1.Em7.ControlNodes".sepaClamp.sequence.status.currentStep = #JOB_11_STEP_01) AND "Unit1.Em7.ControlNodes".sepaClamp.sequence.status.seqActive AND "Unit1.Em7.ControlNodes".sepaClamp."step".transition1[1101] THEN
       "Unit1.Em7.ControlNodes".sepaClamp.sequence.status.nextStep := #JOB_11_STEP_10;
   END_IF;
END_REGION

REGION Network 46: Step[1110] : Clamp Top Open
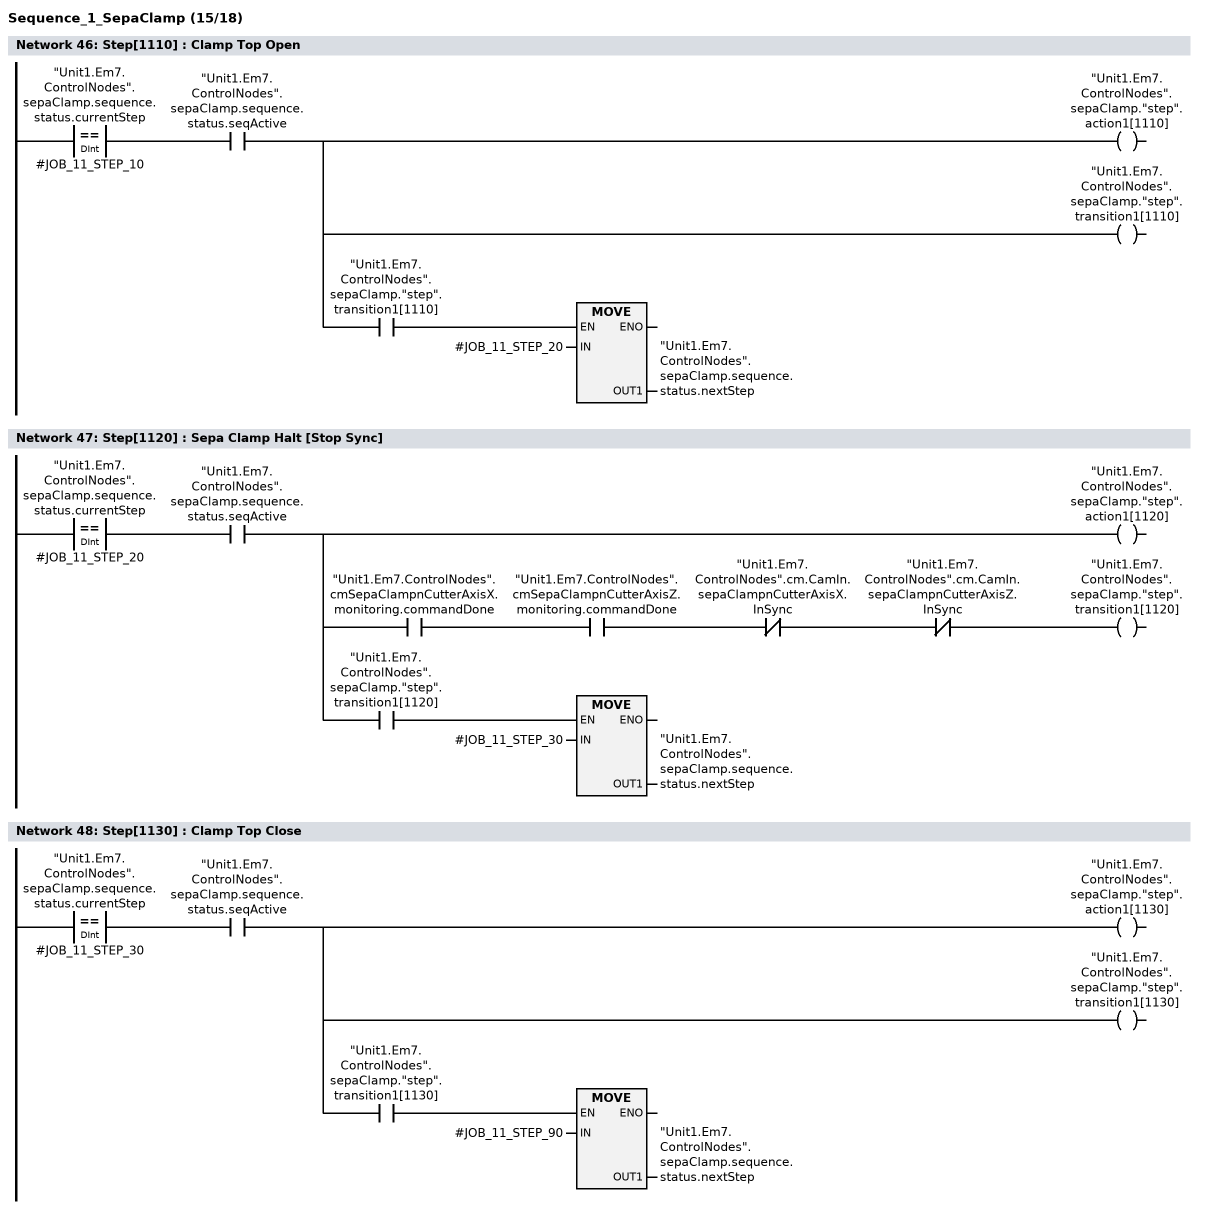
   RUNG wire#powerrail
      { S7_Templates := "SrcType := DInt" } EQ_Contact(in1 := "Unit1.Em7.ControlNodes".sepaClamp.sequence.status.currentStep, in2 := #JOB_11_STEP_10)
      Contact( "Unit1.Em7.ControlNodes".sepaClamp.sequence.status.seqActive )
      wire#w1
      Coil( "Unit1.Em7.ControlNodes".sepaClamp."step".action1[1110] )
   END_RUNG
   RUNG wire#w1
      Coil( "Unit1.Em7.ControlNodes".sepaClamp."step".transition1[1110] )
   END_RUNG
   RUNG wire#w1
      Contact( "Unit1.Em7.ControlNodes".sepaClamp."step".transition1[1110] )
      Move(in := #JOB_11_STEP_20, out1 => "Unit1.Em7.ControlNodes".sepaClamp.sequence.status.nextStep)
   END_RUNG
   // the same network as SCL:
   "Unit1.Em7.ControlNodes".sepaClamp."step".action1[1110] := ("Unit1.Em7.ControlNodes".sepaClamp.sequence.status.currentStep = #JOB_11_STEP_10) AND "Unit1.Em7.ControlNodes".sepaClamp.sequence.status.seqActive;
   "Unit1.Em7.ControlNodes".sepaClamp."step".transition1[1110] := ("Unit1.Em7.ControlNodes".sepaClamp.sequence.status.currentStep = #JOB_11_STEP_10) AND "Unit1.Em7.ControlNodes".sepaClamp.sequence.status.seqActive;
   IF ("Unit1.Em7.ControlNodes".sepaClamp.sequence.status.currentStep = #JOB_11_STEP_10) AND "Unit1.Em7.ControlNodes".sepaClamp.sequence.status.seqActive AND "Unit1.Em7.ControlNodes".sepaClamp."step".transition1[1110] THEN
       "Unit1.Em7.ControlNodes".sepaClamp.sequence.status.nextStep := #JOB_11_STEP_20;
   END_IF;
END_REGION

REGION Network 47: Step[1120] : Sepa Clamp Halt [Stop Sync]
   RUNG wire#powerrail
      { S7_Templates := "SrcType := DInt" } EQ_Contact(in1 := "Unit1.Em7.ControlNodes".sepaClamp.sequence.status.currentStep, in2 := #JOB_11_STEP_20)
      Contact( "Unit1.Em7.ControlNodes".sepaClamp.sequence.status.seqActive )
      wire#w1
      Coil( "Unit1.Em7.ControlNodes".sepaClamp."step".action1[1120] )
   END_RUNG
   RUNG wire#w1
      Contact( "Unit1.Em7.ControlNodes".cmSepaClampnCutterAxisX.monitoring.commandDone )
      Contact( "Unit1.Em7.ControlNodes".cmSepaClampnCutterAxisZ.monitoring.commandDone )
      I_Contact( "Unit1.Em7.ControlNodes".cm.CamIn.sepaClampnCutterAxisX.InSync )
      I_Contact( "Unit1.Em7.ControlNodes".cm.CamIn.sepaClampnCutterAxisZ.InSync )
      Coil( "Unit1.Em7.ControlNodes".sepaClamp."step".transition1[1120] )
   END_RUNG
   RUNG wire#w1
      Contact( "Unit1.Em7.ControlNodes".sepaClamp."step".transition1[1120] )
      Move(in := #JOB_11_STEP_30, out1 => "Unit1.Em7.ControlNodes".sepaClamp.sequence.status.nextStep)
   END_RUNG
   // the same network as SCL:
   "Unit1.Em7.ControlNodes".sepaClamp."step".action1[1120] := ("Unit1.Em7.ControlNodes".sepaClamp.sequence.status.currentStep = #JOB_11_STEP_20) AND "Unit1.Em7.ControlNodes".sepaClamp.sequence.status.seqActive;
   "Unit1.Em7.ControlNodes".sepaClamp."step".transition1[1120] := ("Unit1.Em7.ControlNodes".sepaClamp.sequence.status.currentStep = #JOB_11_STEP_20) AND "Unit1.Em7.ControlNodes".sepaClamp.sequence.status.seqActive AND "Unit1.Em7.ControlNodes".cmSepaClampnCutterAxisX.monitoring.commandDone AND "Unit1.Em7.ControlNodes".cmSepaClampnCutterAxisZ.monitoring.commandDone AND NOT "Unit1.Em7.ControlNodes".cm.CamIn.sepaClampnCutterAxisX.InSync AND NOT "Unit1.Em7.ControlNodes".cm.CamIn.sepaClampnCutterAxisZ.InSync;
   IF ("Unit1.Em7.ControlNodes".sepaClamp.sequence.status.currentStep = #JOB_11_STEP_20) AND "Unit1.Em7.ControlNodes".sepaClamp.sequence.status.seqActive AND "Unit1.Em7.ControlNodes".sepaClamp."step".transition1[1120] THEN
       "Unit1.Em7.ControlNodes".sepaClamp.sequence.status.nextStep := #JOB_11_STEP_30;
   END_IF;
END_REGION

REGION Network 48: Step[1130] : Clamp Top Close
   RUNG wire#powerrail
      { S7_Templates := "SrcType := DInt" } EQ_Contact(in1 := "Unit1.Em7.ControlNodes".sepaClamp.sequence.status.currentStep, in2 := #JOB_11_STEP_30)
      Contact( "Unit1.Em7.ControlNodes".sepaClamp.sequence.status.seqActive )
      wire#w1
      Coil( "Unit1.Em7.ControlNodes".sepaClamp."step".action1[1130] )
   END_RUNG
   RUNG wire#w1
      Coil( "Unit1.Em7.ControlNodes".sepaClamp."step".transition1[1130] )
   END_RUNG
   RUNG wire#w1
      Contact( "Unit1.Em7.ControlNodes".sepaClamp."step".transition1[1130] )
      Move(in := #JOB_11_STEP_90, out1 => "Unit1.Em7.ControlNodes".sepaClamp.sequence.status.nextStep)
   END_RUNG
   // the same network as SCL:
   "Unit1.Em7.ControlNodes".sepaClamp."step".action1[1130] := ("Unit1.Em7.ControlNodes".sepaClamp.sequence.status.currentStep = #JOB_11_STEP_30) AND "Unit1.Em7.ControlNodes".sepaClamp.sequence.status.seqActive;
   "Unit1.Em7.ControlNodes".sepaClamp."step".transition1[1130] := ("Unit1.Em7.ControlNodes".sepaClamp.sequence.status.currentStep = #JOB_11_STEP_30) AND "Unit1.Em7.ControlNodes".sepaClamp.sequence.status.seqActive;
   IF ("Unit1.Em7.ControlNodes".sepaClamp.sequence.status.currentStep = #JOB_11_STEP_30) AND "Unit1.Em7.ControlNodes".sepaClamp.sequence.status.seqActive AND "Unit1.Em7.ControlNodes".sepaClamp."step".transition1[1130] THEN
       "Unit1.Em7.ControlNodes".sepaClamp.sequence.status.nextStep := #JOB_11_STEP_90;
   END_IF;
END_REGION

REGION Network 49: Step[1190] : Job[11] Step End
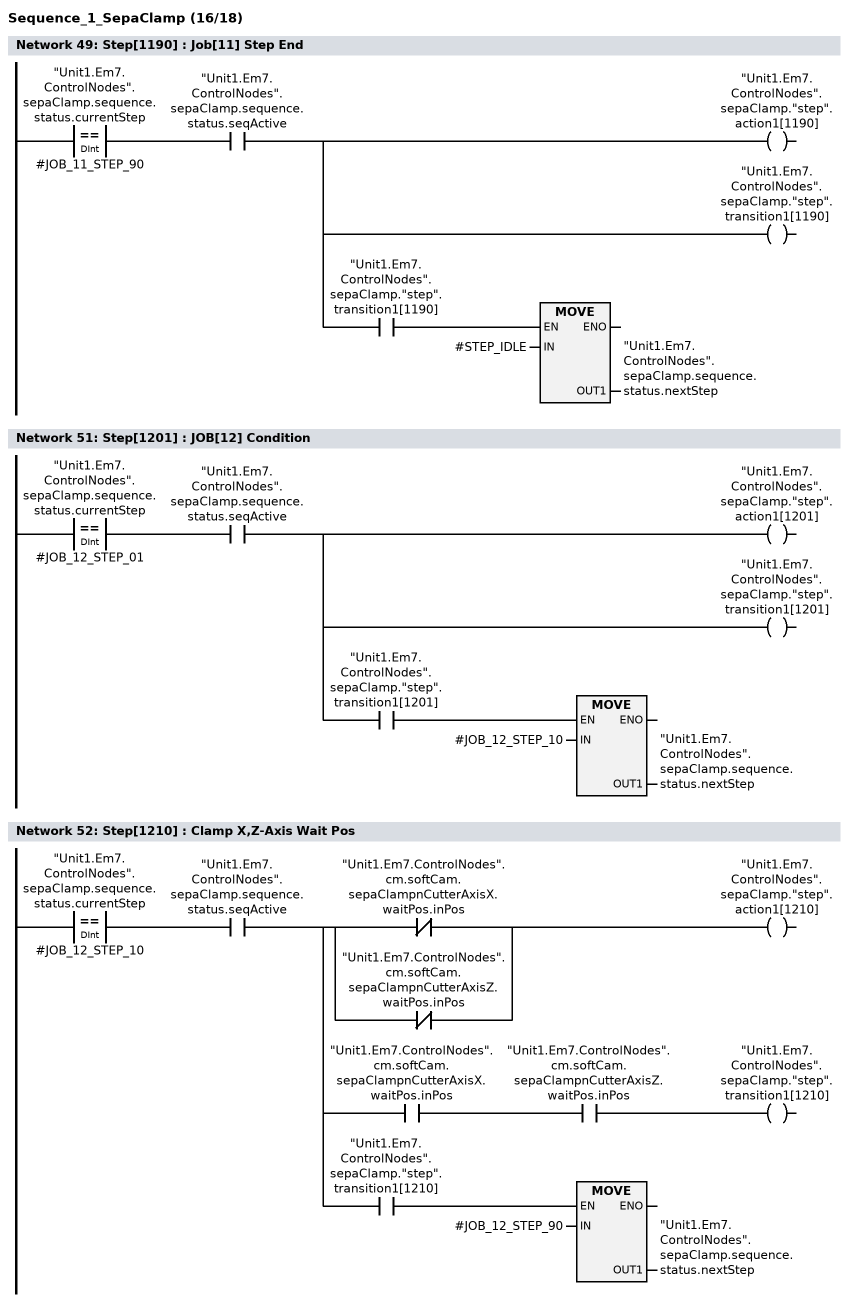
   RUNG wire#powerrail
      { S7_Templates := "SrcType := DInt" } EQ_Contact(in1 := "Unit1.Em7.ControlNodes".sepaClamp.sequence.status.currentStep, in2 := #JOB_11_STEP_90)
      Contact( "Unit1.Em7.ControlNodes".sepaClamp.sequence.status.seqActive )
      wire#w1
      Coil( "Unit1.Em7.ControlNodes".sepaClamp."step".action1[1190] )
   END_RUNG
   RUNG wire#w1
      Coil( "Unit1.Em7.ControlNodes".sepaClamp."step".transition1[1190] )
   END_RUNG
   RUNG wire#w1
      Contact( "Unit1.Em7.ControlNodes".sepaClamp."step".transition1[1190] )
      Move(in := #STEP_IDLE, out1 => "Unit1.Em7.ControlNodes".sepaClamp.sequence.status.nextStep)
   END_RUNG
   // the same network as SCL:
   "Unit1.Em7.ControlNodes".sepaClamp."step".action1[1190] := ("Unit1.Em7.ControlNodes".sepaClamp.sequence.status.currentStep = #JOB_11_STEP_90) AND "Unit1.Em7.ControlNodes".sepaClamp.sequence.status.seqActive;
   "Unit1.Em7.ControlNodes".sepaClamp."step".transition1[1190] := ("Unit1.Em7.ControlNodes".sepaClamp.sequence.status.currentStep = #JOB_11_STEP_90) AND "Unit1.Em7.ControlNodes".sepaClamp.sequence.status.seqActive;
   IF ("Unit1.Em7.ControlNodes".sepaClamp.sequence.status.currentStep = #JOB_11_STEP_90) AND "Unit1.Em7.ControlNodes".sepaClamp.sequence.status.seqActive AND "Unit1.Em7.ControlNodes".sepaClamp."step".transition1[1190] THEN
       "Unit1.Em7.ControlNodes".sepaClamp.sequence.status.nextStep := #STEP_IDLE;
   END_IF;
END_REGION

REGION Network 50: ******************** JOB[12] Unload Return ********************
END_REGION

REGION Network 51: Step[1201] : JOB[12] Condition
   RUNG wire#powerrail
      { S7_Templates := "SrcType := DInt" } EQ_Contact(in1 := "Unit1.Em7.ControlNodes".sepaClamp.sequence.status.currentStep, in2 := #JOB_12_STEP_01)
      Contact( "Unit1.Em7.ControlNodes".sepaClamp.sequence.status.seqActive )
      wire#w1
      Coil( "Unit1.Em7.ControlNodes".sepaClamp."step".action1[1201] )
   END_RUNG
   RUNG wire#w1
      Coil( "Unit1.Em7.ControlNodes".sepaClamp."step".transition1[1201] )
   END_RUNG
   RUNG wire#w1
      Contact( "Unit1.Em7.ControlNodes".sepaClamp."step".transition1[1201] )
      Move(in := #JOB_12_STEP_10, out1 => "Unit1.Em7.ControlNodes".sepaClamp.sequence.status.nextStep)
   END_RUNG
   // the same network as SCL:
   "Unit1.Em7.ControlNodes".sepaClamp."step".action1[1201] := ("Unit1.Em7.ControlNodes".sepaClamp.sequence.status.currentStep = #JOB_12_STEP_01) AND "Unit1.Em7.ControlNodes".sepaClamp.sequence.status.seqActive;
   "Unit1.Em7.ControlNodes".sepaClamp."step".transition1[1201] := ("Unit1.Em7.ControlNodes".sepaClamp.sequence.status.currentStep = #JOB_12_STEP_01) AND "Unit1.Em7.ControlNodes".sepaClamp.sequence.status.seqActive;
   IF ("Unit1.Em7.ControlNodes".sepaClamp.sequence.status.currentStep = #JOB_12_STEP_01) AND "Unit1.Em7.ControlNodes".sepaClamp.sequence.status.seqActive AND "Unit1.Em7.ControlNodes".sepaClamp."step".transition1[1201] THEN
       "Unit1.Em7.ControlNodes".sepaClamp.sequence.status.nextStep := #JOB_12_STEP_10;
   END_IF;
END_REGION

REGION Network 52: Step[1210] : Clamp X,Z-Axis Wait Pos
   RUNG wire#powerrail
      { S7_Templates := "SrcType := DInt" } EQ_Contact(in1 := "Unit1.Em7.ControlNodes".sepaClamp.sequence.status.currentStep, in2 := #JOB_12_STEP_10)
      Contact( "Unit1.Em7.ControlNodes".sepaClamp.sequence.status.seqActive )
      wire#w1
      I_Contact( "Unit1.Em7.ControlNodes".cm.softCam.sepaClampnCutterAxisX.waitPos.inPos )
      wire#w2
      Coil( "Unit1.Em7.ControlNodes".sepaClamp."step".action1[1210] )
   END_RUNG
   RUNG wire#w1
      I_Contact( "Unit1.Em7.ControlNodes".cm.softCam.sepaClampnCutterAxisZ.waitPos.inPos )
   END_RUNG wire#w2
   RUNG wire#w1
      Contact( "Unit1.Em7.ControlNodes".cm.softCam.sepaClampnCutterAxisX.waitPos.inPos )
      Contact( "Unit1.Em7.ControlNodes".cm.softCam.sepaClampnCutterAxisZ.waitPos.inPos )
      Coil( "Unit1.Em7.ControlNodes".sepaClamp."step".transition1[1210] )
   END_RUNG
   RUNG wire#w1
      Contact( "Unit1.Em7.ControlNodes".sepaClamp."step".transition1[1210] )
      Move(in := #JOB_12_STEP_90, out1 => "Unit1.Em7.ControlNodes".sepaClamp.sequence.status.nextStep)
   END_RUNG
   // the same network as SCL:
   #_w1 := ("Unit1.Em7.ControlNodes".sepaClamp.sequence.status.currentStep = #JOB_12_STEP_10) AND "Unit1.Em7.ControlNodes".sepaClamp.sequence.status.seqActive;
   "Unit1.Em7.ControlNodes".sepaClamp."step".action1[1210] := #_w1 AND (NOT "Unit1.Em7.ControlNodes".cm.softCam.sepaClampnCutterAxisX.waitPos.inPos OR NOT "Unit1.Em7.ControlNodes".cm.softCam.sepaClampnCutterAxisZ.waitPos.inPos);
   "Unit1.Em7.ControlNodes".sepaClamp."step".transition1[1210] := #_w1 AND "Unit1.Em7.ControlNodes".cm.softCam.sepaClampnCutterAxisX.waitPos.inPos AND "Unit1.Em7.ControlNodes".cm.softCam.sepaClampnCutterAxisZ.waitPos.inPos;
   IF #_w1 AND "Unit1.Em7.ControlNodes".sepaClamp."step".transition1[1210] THEN
       "Unit1.Em7.ControlNodes".sepaClamp.sequence.status.nextStep := #JOB_12_STEP_90;
   END_IF;
END_REGION

REGION Network 53: Step[1290] : Job[12] Step End
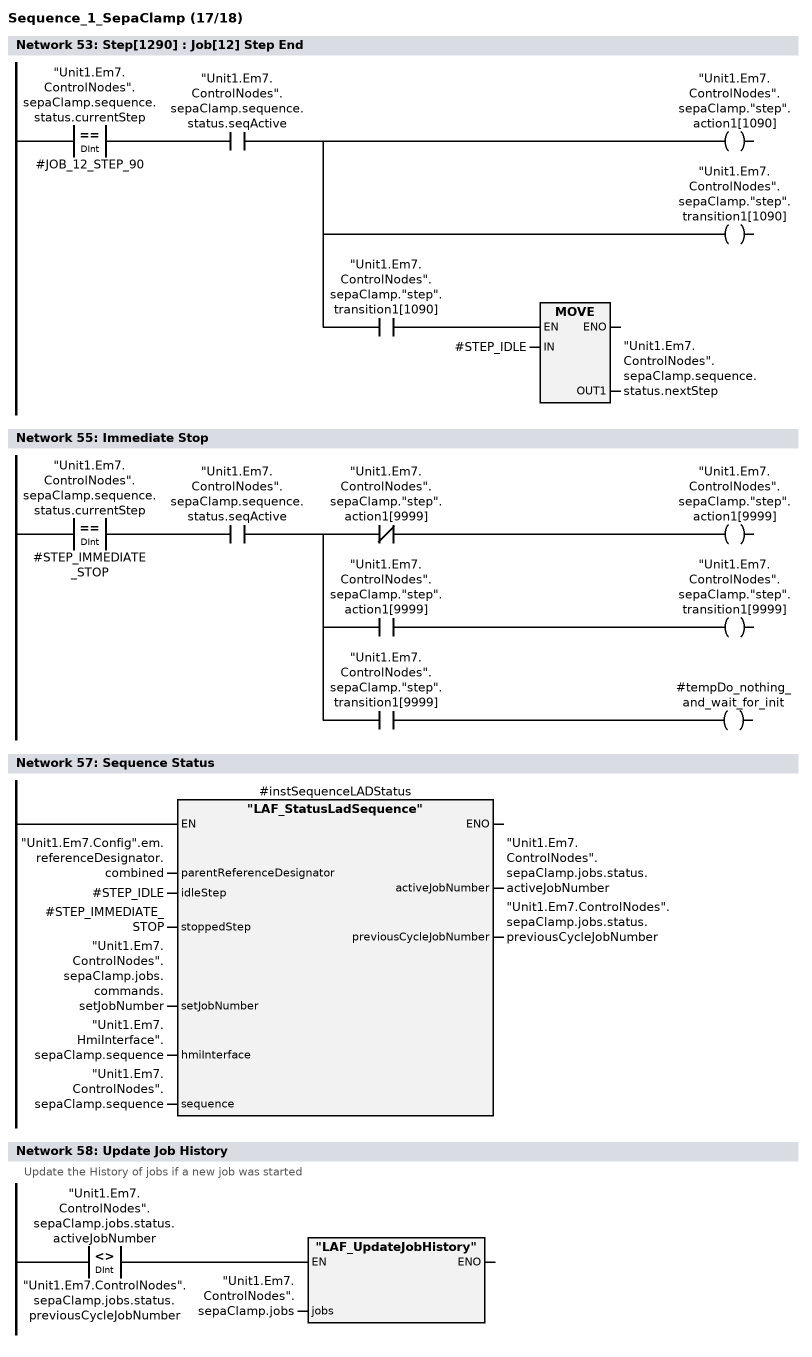
   RUNG wire#powerrail
      { S7_Templates := "SrcType := DInt" } EQ_Contact(in1 := "Unit1.Em7.ControlNodes".sepaClamp.sequence.status.currentStep, in2 := #JOB_12_STEP_90)
      Contact( "Unit1.Em7.ControlNodes".sepaClamp.sequence.status.seqActive )
      wire#w1
      Coil( "Unit1.Em7.ControlNodes".sepaClamp."step".action1[1090] )
   END_RUNG
   RUNG wire#w1
      Coil( "Unit1.Em7.ControlNodes".sepaClamp."step".transition1[1090] )
   END_RUNG
   RUNG wire#w1
      Contact( "Unit1.Em7.ControlNodes".sepaClamp."step".transition1[1090] )
      Move(in := #STEP_IDLE, out1 => "Unit1.Em7.ControlNodes".sepaClamp.sequence.status.nextStep)
   END_RUNG
   // the same network as SCL:
   "Unit1.Em7.ControlNodes".sepaClamp."step".action1[1090] := ("Unit1.Em7.ControlNodes".sepaClamp.sequence.status.currentStep = #JOB_12_STEP_90) AND "Unit1.Em7.ControlNodes".sepaClamp.sequence.status.seqActive;
   "Unit1.Em7.ControlNodes".sepaClamp."step".transition1[1090] := ("Unit1.Em7.ControlNodes".sepaClamp.sequence.status.currentStep = #JOB_12_STEP_90) AND "Unit1.Em7.ControlNodes".sepaClamp.sequence.status.seqActive;
   IF ("Unit1.Em7.ControlNodes".sepaClamp.sequence.status.currentStep = #JOB_12_STEP_90) AND "Unit1.Em7.ControlNodes".sepaClamp.sequence.status.seqActive AND "Unit1.Em7.ControlNodes".sepaClamp."step".transition1[1090] THEN
       "Unit1.Em7.ControlNodes".sepaClamp.sequence.status.nextStep := #STEP_IDLE;
   END_IF;
END_REGION

REGION Network 54: *************** IMMEDIATE STOP **************************
END_REGION

REGION Network 55: Immediate Stop
   RUNG wire#powerrail
      { S7_Templates := "SrcType := DInt" } EQ_Contact(in1 := "Unit1.Em7.ControlNodes".sepaClamp.sequence.status.currentStep, in2 := #STEP_IMMEDIATE_STOP)
      Contact( "Unit1.Em7.ControlNodes".sepaClamp.sequence.status.seqActive )
      wire#w1
      I_Contact( "Unit1.Em7.ControlNodes".sepaClamp."step".action1[9999] )
      Coil( "Unit1.Em7.ControlNodes".sepaClamp."step".action1[9999] )
   END_RUNG
   RUNG wire#w1
      Contact( "Unit1.Em7.ControlNodes".sepaClamp."step".action1[9999] )
      Coil( "Unit1.Em7.ControlNodes".sepaClamp."step".transition1[9999] )
   END_RUNG
   RUNG wire#w1
      Contact( "Unit1.Em7.ControlNodes".sepaClamp."step".transition1[9999] )
      Coil( #tempDo_nothing_and_wait_for_init )
   END_RUNG
   // the same network as SCL:
   #_w1 := ("Unit1.Em7.ControlNodes".sepaClamp.sequence.status.currentStep = #STEP_IMMEDIATE_STOP) AND "Unit1.Em7.ControlNodes".sepaClamp.sequence.status.seqActive;
   "Unit1.Em7.ControlNodes".sepaClamp."step".action1[9999] := #_w1 AND NOT "Unit1.Em7.ControlNodes".sepaClamp."step".action1[9999];
   "Unit1.Em7.ControlNodes".sepaClamp."step".transition1[9999] := #_w1 AND "Unit1.Em7.ControlNodes".sepaClamp."step".action1[9999];
   #tempDo_nothing_and_wait_for_init := #_w1 AND "Unit1.Em7.ControlNodes".sepaClamp."step".transition1[9999];
END_REGION

REGION Network 56: *************** Status updates **************************
END_REGION

REGION Network 57: Sequence Status
   RUNG wire#powerrail
      #instSequenceLADStatus(parentReferenceDesignator := "Unit1.Em7.Config".em.referenceDesignator.combined, idleStep := #STEP_IDLE, stoppedStep := #STEP_IMMEDIATE_STOP, setJobNumber := "Unit1.Em7.ControlNodes".sepaClamp.jobs.commands.setJobNumber, hmiInterface := "Unit1.Em7.HmiInterface".sepaClamp.sequence, sequence := "Unit1.Em7.ControlNodes".sepaClamp.sequence, activeJobNumber => "Unit1.Em7.ControlNodes".sepaClamp.jobs.status.activeJobNumber, previousCycleJobNumber => "Unit1.Em7.ControlNodes".sepaClamp.jobs.status.previousCycleJobNumber)
   END_RUNG
   // the same network as SCL:
   #instSequenceLADStatus(parentReferenceDesignator := "Unit1.Em7.Config".em.referenceDesignator.combined,   // "LAF_StatusLadSequence"
                          idleStep := #STEP_IDLE,
                          stoppedStep := #STEP_IMMEDIATE_STOP,
                          setJobNumber := "Unit1.Em7.ControlNodes".sepaClamp.jobs.commands.setJobNumber,
                          hmiInterface := "Unit1.Em7.HmiInterface".sepaClamp.sequence,
                          sequence := "Unit1.Em7.ControlNodes".sepaClamp.sequence,
                          activeJobNumber => "Unit1.Em7.ControlNodes".sepaClamp.jobs.status.activeJobNumber,
                          previousCycleJobNumber => "Unit1.Em7.ControlNodes".sepaClamp.jobs.status.previousCycleJobNumber);
END_REGION

REGION Network 58: Update Job History
   // Update the History of jobs if a new job was started
   RUNG wire#powerrail
      { S7_Templates := "SrcType := DInt" } NE_Contact(in1 := "Unit1.Em7.ControlNodes".sepaClamp.jobs.status.activeJobNumber, in2 := "Unit1.Em7.ControlNodes".sepaClamp.jobs.status.previousCycleJobNumber)
      "LAF_UpdateJobHistory"(jobs := "Unit1.Em7.ControlNodes".sepaClamp.jobs)
   END_RUNG
   // the same network as SCL:
   IF "Unit1.Em7.ControlNodes".sepaClamp.jobs.status.activeJobNumber <> "Unit1.Em7.ControlNodes".sepaClamp.jobs.status.previousCycleJobNumber THEN
       "LAF_UpdateJobHistory"(jobs := "Unit1.Em7.ControlNodes".sepaClamp.jobs);
   END_IF;
END_REGION

REGION Network 59: Output steps as String
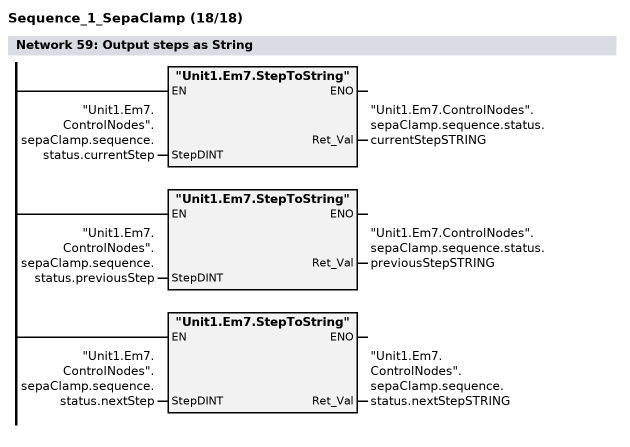
   RUNG wire#powerrail
      "Unit1.Em7.StepToString"(StepDINT := "Unit1.Em7.ControlNodes".sepaClamp.sequence.status.currentStep, Ret_Val => "Unit1.Em7.ControlNodes".sepaClamp.sequence.status.currentStepSTRING)
   END_RUNG
   RUNG wire#powerrail
      "Unit1.Em7.StepToString"(StepDINT := "Unit1.Em7.ControlNodes".sepaClamp.sequence.status.previousStep, Ret_Val => "Unit1.Em7.ControlNodes".sepaClamp.sequence.status.previousStepSTRING)
   END_RUNG
   RUNG wire#powerrail
      "Unit1.Em7.StepToString"(StepDINT := "Unit1.Em7.ControlNodes".sepaClamp.sequence.status.nextStep, Ret_Val => "Unit1.Em7.ControlNodes".sepaClamp.sequence.status.nextStepSTRING)
   END_RUNG
   // the same network as SCL:
   "Unit1.Em7.ControlNodes".sepaClamp.sequence.status.currentStepSTRING := "Unit1.Em7.StepToString"(StepDINT := "Unit1.Em7.ControlNodes".sepaClamp.sequence.status.currentStep);
   "Unit1.Em7.ControlNodes".sepaClamp.sequence.status.previousStepSTRING := "Unit1.Em7.StepToString"(StepDINT := "Unit1.Em7.ControlNodes".sepaClamp.sequence.status.previousStep);
   "Unit1.Em7.ControlNodes".sepaClamp.sequence.status.nextStepSTRING := "Unit1.Em7.StepToString"(StepDINT := "Unit1.Em7.ControlNodes".sepaClamp.sequence.status.nextStep);
END_REGION
END_FUNCTION_BLOCK
